# B&R Automation Studio project NAINV104C00R8L515F00 (part 26)

#### Act_Background_Action.st - not listed in the package file held
```iecst
(** 2021-08-01 **)
ACTION Act_Background_Action:
	//Action function
//testing funciton
	IF EDGEPOS(bSimBrdInZone1) THEN
		tyHermesBoardAvailableAttribAddr.udiProductTypeId := p_ProdRcpCurrRcp0Nm;
		tyHermesBoardAvailableAttribAddr.udiWidth  := p_ProdRcpCurrRcp0Width;
		fHermesGenerateBrdAvlDat(ADR(a_tyHermesBrdAvlData[1]),tyHermesBoardAvailableAttribAddr);
		fHermesAddEditAttribBrdAvlDat(ADR(a_tyHermesBrdAvlData[1]),'Action',sSelectedActtoUpdate);
		bSimBrdInZone1 := FALSE;
	END_IF
	IF EDGEPOS(bSimBrdInZone2) THEN
		tyHermesBoardAvailableAttribAddr.udiProductTypeId := p_ProdRcpCurrRcp0Nm;
		tyHermesBoardAvailableAttribAddr.udiWidth  := p_ProdRcpCurrRcp0Width;
		fHermesGenerateBrdAvlDat(ADR(a_tyHermesBrdAvlData[2]),tyHermesBoardAvailableAttribAddr);
		fHermesAddEditAttribBrdAvlDat(ADR(a_tyHermesBrdAvlData[2]),'Action',sSelectedActtoUpdate);
		bSimBrdInZone2 := FALSE;
	END_IF
	IF EDGEPOS(bSimBrdInZone3) THEN
		tyHermesBoardAvailableAttribAddr.udiProductTypeId := p_ProdRcpCurrRcp0Nm;
		tyHermesBoardAvailableAttribAddr.udiWidth  := p_ProdRcpCurrRcp0Width;
		fHermesGenerateBrdAvlDat(ADR(a_tyHermesBrdAvlData[3]),tyHermesBoardAvailableAttribAddr);
		fHermesAddEditAttribBrdAvlDat(ADR(a_tyHermesBrdAvlData[3]),'Action',sSelectedActtoUpdate);
		bSimBrdInZone3 := FALSE;
	END_IF
//	IF EDGEPOS(bSimSearch) THEN
//		testresult1 := fHermesSrchAttribValueBrdAvlDat(ADR(a_tyHermesBrdAvlData[1]),'Action',ADR(sAttribReadValue));
//	END_IF
//	IF EDGEPOS(bSimDelete) THEN
//		testresult2 := fHermesDeleteAttribBrdAvlDat(ADR(a_tyHermesBrdAvlData[1]),'Action');
//	END_IF

	IF EDGEPOS(bSimShiftBoardFoward) THEN
		memmove(ADR(a_tyHermesBrdAvlData[endpos]),ADR(a_tyHermesBrdAvlData[startpos]),SIZEOF(a_tyHermesBrdAvlData[startpos]));
		memset(ADR(a_tyHermesBrdAvlData[startpos]),0,SIZEOF(a_tyHermesBrdAvlData[startpos]));
		memmove(ADR(a_bLinkOpsGConvHvBrd[endpos]),ADR(a_bLinkOpsGConvHvBrd[startpos]),SIZEOF(a_bLinkOpsGConvHvBrd[startpos]));
		memset(ADR(a_bLinkOpsGConvHvBrd[startpos]),0,SIZEOF(a_bLinkOpsGConvHvBrd[startpos]));
	END_IF
	IF EDGEPOS(bSimClear) THEN
		memset(ADR(a_tyHermesBrdAvlData[dltpos]),0,SIZEOF(a_tyHermesBrdAvlData[dltpos]));
	END_IF
//end of testing

//	In state Below
//	Zone[supported action]    0 | 1 | 2
//	Brd(supported action)    A | B | C

	FOR usiZone := usiZoneSupported TO 1 BY -1 DO
		//assiging action
		//update for next machine or zone action
		IF  NOT(a_bUIZonePause[usiZone]) THEN
			a_bBlkDSForAction[usiZone] := FALSE;
			a_bUIPromptActionSelect[usiZone] := FALSE;
		ELSE
			a_bBlkDSForAction[usiZone] := TRUE;
			IF EDGEPOS(a_bOpsDsStandByStep[usiZone]) THEN
				a_bUIPromptActionSelect[usiZone] := TRUE ;
			END_IF

			IF EDGENEG(a_bUIPromptActionSelect[usiZone])  THEN
				a_bUIZonePause[usiZone] := FALSE;
				udiSelectedModtoUpt := a_eModSelectedforCurrZone[usiZone];
				sSelectedActtoUpdate := UDINT_TO_STRING(udiSelectedModtoUpt);
				fHermesAddEditAttribBrdAvlDat(ADR(a_tyHermesBrdAvlData[usiZone]),'Action',sSelectedActtoUpdate);

			END_IF
		END_IF

		//switch the mod for that zone as soon as possible
		//below for preparing action for unoccupied zone starting from right most

		//1)block zone occurred to prevent the middle zone stop reacting to the pending board which does not meet its supported action
		//2)not until the estimated board reach the supported zone, the other left zone will not assigned with action
		//3)compare the leftblock , if reservation zone and occupied zone happened at same time, choose the leftmost zone
		IF usiZone = usiZoneSupported THEN
			usiLeftmostBlockedZone := usiZone;
		ELSIF usiZone < usiLeftmostBlockedZone THEN
			usiLeftmostBlockedZone := usiZone; //check the left block zone
		END_IF

		IF a_bLinkOpsGConvStepInitDone[usiZone] THEN
			IF NOT(a_bLinkOpsGConvHvBrd[usiZone]) THEN
				memset(ADR(a_tyActionReservedForZone[usiZone]),0,SIZEOF(a_tyActionReservedForZone[usiZone]));
				IF usiLeftmostBlockedZone <> 0 THEN //occured there is zone reserved or occupied at zone 1
					FOR usiBrdZone := usiLeftmostBlockedZone TO 1 BY -1 DO
						IF a_bLinkOpsGConvHvBrd[usiBrdZone] THEN
							IF (usiBrdZone-1) < usiZone THEN
								usiLeftmostBlockedZone :=  usiBrdZone; //current board position as limit
							END_IF
							iActionAttributeIdx := fHermesSrchAttribValueBrdAvlDat(ADR(a_tyHermesBrdAvlData[usiBrdZone]),'Action',ADR(sAttribReadValue));
							IF iActionAttributeIdx <> -1 THEN
								iActionOnBrd := STRING_TO_INT(sAttribReadValue);
								IF iActionOnBrd <> 0 AND (1 <= iActionOnBrd  AND iActionOnBrd <= usiMaxActionSupported )THEN
									IF tbActionSupportedByZone[usiZone,iActionOnBrd] THEN
										fHermesSrchAttribValueBrdAvlDat(ADR(a_tyHermesBrdAvlData[usiBrdZone]),'BoardId',ADR(sAttribReadValue));
										//the zone pro-react to action on board
										IF (usiBrdZone-1) < usiZone THEN
											usiLeftmostBlockedZone := usiBrdZone -1; //choose board starting from left side
										END_IF
										a_tyActionReservedForZone[usiZone].iAction := iActionOnBrd; //found support on this zone
										a_tyActionReservedForZone[usiZone].iAttributeIdx := iActionAttributeIdx +1;
										a_tyActionReservedForZone[usiZone].sBoardId := sAttribReadValue;
										EXIT;
									END_IF
								END_IF
							END_IF
							IF a_tyActionReservedForZone[usiZone].iAction <> iActionOnBrd OR iActionOnBrd = 0 THEN
								EXIT; //when non-supported board stuck at middle then do no consider further
							END_IF
						END_IF
					END_FOR
				END_IF
			ELSE // if have board
				IF (usiZone -1) < usiLeftmostBlockedZone THEN
					usiLeftmostBlockedZone := usiZone -1;
				END_IF
				//update when action completed
				fHermesSrchAttribValueBrdAvlDat(ADR(a_tyHermesBrdAvlData[usiZone]),'BoardId',ADR(sAttribReadValue));
				IF a_tyActionReservedForZone[usiZone].iAction <> 0 AND sAttribReadValue =  a_tyActionReservedForZone[usiZone].sBoardId THEN
					IF a_tyActionReservedForZone[usiZone].bActionCompl THEN
						a_tyHermesBrdAvlData[usiZone].a_tyXMLTableDataBrdAvl[a_tyActionReservedForZone[usiZone].iAttributeIdx].sValue	:= '0';
					END_IF
				ELSE //refind an action for the board in current zone
					memset(ADR(a_tyActionReservedForZone[usiZone]),0,SIZEOF(a_tyActionReservedForZone[usiZone]));
					iActionAttributeIdx := fHermesSrchAttribValueBrdAvlDat(ADR(a_tyHermesBrdAvlData[usiZone]),'Action',ADR(sAttribReadValue));
					IF iActionAttributeIdx <> -1 THEN
						iActionOnBrd := STRING_TO_INT(sAttribReadValue);
						IF iActionOnBrd <> 0 AND (1 <= iActionOnBrd  AND iActionOnBrd <= usiMaxActionSupported )THEN
							IF tbActionSupportedByZone[usiZone,iActionOnBrd] THEN
								//react
								fHermesSrchAttribValueBrdAvlDat(ADR(a_tyHermesBrdAvlData[usiZone]),'BoardId',ADR(sAttribReadValue));
								a_tyActionReservedForZone[usiZone].iAction := iActionOnBrd; //found support on this zone
								a_tyActionReservedForZone[usiZone].iAttributeIdx := iActionAttributeIdx +1;
								a_tyActionReservedForZone[usiZone].sBoardId := sAttribReadValue;
								EXIT;
							END_IF
						END_IF
					END_IF
				END_IF
			END_IF

		END_IF

	END_FOR

END_ACTION
```

### USHermes.var - Change By Project
```iecst
(*2020-09-10*)
(**)
(*Action & State & Status*)
VAR
	p_USHermesStat : UDINT;
	p_USHermesStatus : UDINT;
	p_USHermesStatTxt : UDINT;
END_VAR
(**)
(*Alarm*)
VAR
	p_USHermesAlmData : UDINT;
	p_USHermesAlmData1 : UDINT;
	p_USHermesAlmData2 : UDINT;
	p_USHermesAlmData3 : UDINT;
	p_USHermesAlmData4 : UDINT;
	p_USHermesAlmData5 : UDINT;
	p_USHermesInfoData : UDINT;
END_VAR
(**)
(*Output*)
VAR
	p_USHermesTableDataBrdAvl : UDINT;
	p_USHermesTableDataBrdAvlTtlIdx : UDINT;
	p_USHermesConnected : UDINT;
	p_USHermesHandshakeDone : UDINT;
	p_USHermesAccDataReq : UDINT;
	p_USHermesOverWriteSlt : UDINT;
	p_USHermesOverWriteWidth : UDINT;
	p_USHermesReqRecipeNm : UDINT;
	p_USHermesReqWidthInUM : UDINT;
	p_USHermesReqMinSltValue : UDINT;
	p_USHermesReqMaxSltValue : UDINT;
	p_USHermesReqPitch : UDINT;
	p_USHermesUSRdy : UDINT;
	p_USHermesDSRdy : UDINT;
	p_USHermesUSGdRdy : UDINT;
	p_USHermesDSGdRdy : UDINT;
	p_USHermesTransporting : UDINT;
	p_USHermesStopTransport : UDINT;
	p_USHermesBlkUS : UDINT;
	p_USHermesInternalSnd : UDINT;
	p_USHermesAccDataMnl : UDINT;
	p_USHermesStopTransportSnd : UDINT;
	p_USHermestyBoardAvailable : UDINT;
	p_USHermesBoardArrivedData : UDINT;
	p_USHermesRcvBoardInfoOk : UDINT;
	p_USHermesRcvbBoardInfoIncompl : UDINT;
	p_USHermesBoardInfoData : UDINT;
	p_USHermesCommandParam : UDINT;
	p_USHermesReverseDSSendBFId : UDINT;
	p_USHermesProcessRouteTrigger : UDINT;
	p_USHermesAction : UDINT;
	p_USHermesBrdForecastRcv : UDINT;
	p_USHermesBoardAvailableRcved : UDINT;
	p_USHermesStopTransportSent : UDINT;
	p_USHermesStopTransportSentMsg : UDINT;
	p_USHermesBrdForecast : UDINT;
END_VAR
```

### Program Logical/Hermes/USHermes (IEC, version 1.00.0) - 1.00.0 - NtHermes v5.00.0 , NtTCP v5.00.0 , NtMessage v5.00.0

#### Init.st - Change By Project
```iecst
(** 2020-09-10 **)
PROGRAM _INIT

	(* Always Change If Project Change *)

	//Pass Address To Global Address For External Use
	//Action, State & Status
	p_USHermesStat		:= ADR(eStat);
	p_USHermesStatus	:= ADR(eMainStatus);
	p_USHermesStatTxt	:= ADR(sStatTxt);

	//Alarm
	p_USHermesAlmData	:= ADR(tyAlmData);
	p_USHermesAlmData1	:= ADR(tyAlmData1);
	p_USHermesAlmData2	:= ADR(tyAlmData2);
	p_USHermesAlmData3	:= ADR(tyAlmData3);
	p_USHermesAlmData4	:= ADR(tyAlmData4);
	p_USHermesAlmData5	:= ADR(tyAlmData5);
	p_USHermesInfoData	:= ADR(tyInfoData);

	//Output
	p_USHermesTableDataBrdAvl		:= ADR(a_tyXMLTableDataBrdAvl);
	p_USHermesTableDataBrdAvlTtlIdx	:= ADR(iXMLTableDataBrdAvlTtlIdx);
	p_USHermesConnected				:= ADR(bConnected);
	p_USHermesHandshakeDone			:= ADR(bHandshakeDone);
	p_USHermesAccDataReq			:= ADR(bAccDataReq);
	p_USHermesOverWriteSlt			:= ADR(bOverWriteSlt);
	p_USHermesOverWriteWidth		:= ADR(bOverWriteWidth);
	p_USHermesReqRecipeNm			:= ADR(sReqRecipeNm);
	p_USHermesReqWidthInUM			:= ADR(diReqWidthInUM);
	p_USHermesReqMinSltValue		:= ADR(diReqMinSltValue);
	p_USHermesReqMaxSltValue		:= ADR(diReqMaxSltValue);
	p_USHermesReqPitch				:= ADR(diReqPitch);
	p_USHermesUSRdy					:= ADR(bUSRdy);
	p_USHermesDSRdy					:= ADR(bDSRdy);
	p_USHermesUSGdRdy				:= ADR(bUSGdRdy);
	p_USHermesDSGdRdy				:= ADR(bDSGdRdy);
	p_USHermesTransporting			:= ADR(bTransporting);
	p_USHermesStopTransport			:= ADR(bStopTransport);
	p_USHermesBlkUS					:= ADR(bBlkUS);
	p_USHermesInternalSnd			:= ADR(sInternalSnd);
	p_USHermesAccDataMnl			:= ADR(bAccDataMnl);
	p_USHermesStopTransportSnd 		:= ADR(bStopTransportSnd);

	p_USHermestyBoardAvailable		:= ADR(tyBoardAvailableRcv);
	p_USHermesRcvBoardInfoOk        := ADR(bRcvBoardInfoOk);
	p_USHermesRcvbBoardInfoIncompl  := ADR(bRcvBoardInfoIncompl);
	p_USHermesBoardInfoData         := ADR(tySendBoardInfoAcc); //Pass "SendBoardInfo" data for DSHermes "BoardAvailable", for inserted PCB
	p_USHermesBoardArrivedData		:= ADR(tyBoardArrivedInfo); //"BoardArrived" data for SupervisoryHermes

	//command

	p_USHermesCommandParam			:= ADR(tyCommandParam);

	//Calling  on Reverse DS
	p_USHermesReverseDSSendBFId		:= ADR(bReverseDSSndBfWBrdID);
	p_USHermesProcessRouteTrigger	:= ADR(bTriggerUpdateRoute);

	//Action
	p_USHermesAction				:= ADR(iAction);

	//p_USHermesSwitchtoReverseReceive 	:= ADR(bSwitchtoReverseReceive);
	(* Always Change If Project Change *)

	p_USHermesBrdForecast			:= ADR(tyBoardForecastRcv);
	p_USHermesBrdForecastRcv 		:= ADR(bBrdForecastRcv);
	p_USHermesStopTransportSent    	:= ADR(bStopTransportSent);
	p_USHermesStopTransportSentMsg  := ADR(tyStopTransport);
	p_USHermesBoardAvailableRcved   :=ADR(bBoardAvailableRcved);
END_PROGRAM
```

#### Act_InitGlobal.st - Change By Project
```iecst
(** 2019-06-28 **)
ACTION Act_InitGlobal:

	(* Always Change If Project Change *)

	//Pass Data To Link
	p_bLinkStartupRun ACCESS p_StartupRun;
	p_eLinkMcParamUSCommMod ACCESS p_McParamUSCommMod;

	p_eLinkConvDir ACCESS p_NtParamProjConvDir;
	p_bLinkDILeftSen ACCESS p_DIConvLftSen;
	p_bLinkDIRightSen ACCESS p_DIConvRgtSen;

	p_bLinkOpsInvertStepInitDone ACCESS p_OpsInvertStepInitDone;
	p_bLinkOpsRun ACCESS p_OpsRun;

	//Pass Data To Internal Use
	p_udiRstErr ACCESS p_RstErrReset;
	p_bPrep ACCESS p_NtParamHermesPrep;
	p_tyParam ACCESS p_HermesUSParam1;
	p_sIPAddr ACCESS p_HWInfoIPAddr;
	p_tyDTStructure ACCESS p_TimeCurrDTStruct;
	p_dtCurrDT ACCESS p_TimeCurrDT;
	p_sMcId ACCESS p_McParamMcNm;
	p_sRecipeNm ACCESS p_ProdRcpCurrRcp0Nm;
	p_diWidthInUM ACCESS p_ProdRcpCurrRcp0Width;
	p_udiAliveIdleTimeInSec ACCESS p_NtParamUSHermesAliveTmInSec;
	p_tConnTimeOut ACCESS p_NtParamUSHermesConnTO;
	p_diTransferInTO ACCESS p_McParamTranInErrDlyTm;
	p_bInterruptSen ACCESS p_DIConvLftSen;
	p_bOpsRun ACCESS p_OpsRun;
	p_udiFileKeepDay ACCESS p_NtParamUSHermesFileKeepDay;
	p_sProgNm ACCESS p_NtParamUSHermesProgNm;
	p_bNtSettingsLoadDone ACCESS p_StartupNtSettingsLoadDone;
	p_bAccDataRdy ACCESS p_USHermesUSRdy;
	p_sRmtMcId ACCESS p_RmtHermesCurrentConfMcId;
	p_bRmtPrep ACCESS p_NtParamHermesRmtPrep;
	p_bRmtEn ACCESS p_McParamHermesRmtEn;
	pa_tyProdRcpList ACCESS p_ProdRcpCurrList;
	p_tyProdRcpCurrRcp ACCESS p_ProdRcpCurrRcp0;
	p_bMcParamMnlAccData ACCESS p_McParamMnlAccDat;
	p_bUIAccData ACCESS p_UIProdAccData;

	pa_tyHermesDSParam ACCESS pa_HermesDSParam;

	p_bHermesSwitchtoRvrseTransport ACCESS p_HermesSwitchtoReverseTransport;//p_USHermes2SwitchtoReverseRcv;
	//Query Board Info
	p_bTransportFinished ACCESS p_DSHermesTransportFinish ;
	p_bQueryBoardInfo ACCESS p_UIQueryBoardInfo;
	p_bManualInsertZoneHvBrd ACCESS p_ConvHvBrd; //insert zone (can input conv or ouput conv)
	p_bManualInsertEndSen ACCESS p_DIConvRgtSen;
	p_bConvHvBrd ACCESS p_ConvHvBrd; //first zone
	//Reverse Machine Ready
	//p_bReceiveReverseUSMcRdy ACCESS p_DSHermes2RcvReverseUSMcRdy;

	(* Always Change If Project Change *)

END_ACTION
```

#### InputRef_Link.var - Change By Project
```iecst
(*2019-06-04*)
(**)
VAR
	p_bLinkStartupRun : REFERENCE TO BOOL;
	p_eLinkMcParamUSCommMod : REFERENCE TO eMcSetCommMod;
	bHermesRun : BOOL;
	bHermesStop : BOOL;
END_VAR
(**)
VAR
	p_eLinkConvDir : REFERENCE TO eConvDir;
	p_bLinkDILeftSen : REFERENCE TO BOOL;
	p_bLinkDIRightSen : REFERENCE TO BOOL;
	pa_tyLinkProdRcpList : REFERENCE TO ARRAY[1..c_udiProdRcpMax] OF tyProdRcpParam;
	p_tyLinkProdRcpCurrRcp : REFERENCE TO tyProdRcpParam;
	p_bLinkMcParamMnlAccData : REFERENCE TO BOOL;
	p_bLinkOpsStop : REFERENCE TO BOOL;
	p_bLinkUIAccData : REFERENCE TO BOOL;
	sWidthInUMTemp : STRING[80];
END_VAR
(**)
VAR
	p_bLinkConvHvBrd : REFERENCE TO BOOL;
	p_bLinkOpsRun : REFERENCE TO BOOL;
	p_bLinkOpsInvertStepInitDone : REFERENCE TO BOOL;
END_VAR
(**)
VAR
	fbDlyTmr : TON := (PT:=T#5s);
	fbDeleteLogTmr : TON := (PT:=T#24h);
END_VAR
```

#### Act_LinkEn.st - Change By Project
```iecst
(** 2019-03-15 **)
ACTION Act_LinkEn:

	//Link bPrep, bEn & bDis

END_ACTION
```

#### Act_Link.st - Change By Project
```iecst
(** 2019-06-04 **)
ACTION Act_Link:

	//Receive Alive Time
	p_tyParam.tRcvAlive	:= p_tyParam.tSndAlive * 2;

	//Transfer Complete
	IF (p_eLinkConvDir = ConvDirLToR) OR (p_eLinkConvDir = ConvDirLToL) THEN
		p_bRcvCompl	:= EDGENEG(p_bLinkDILeftSen);
	ELSE
		p_bRcvCompl	:= EDGENEG(p_bLinkDIRightSen);
	END_IF

	//Ready Receive
	p_bRdyRcv ACCESS p_OpsInvertStepUSCommTmr;

	//Ready Transport
	p_bRdyTransport	:= TRUE;

	//Accept New Recipe Condition
	p_bAccNewRcpCond	:= p_bLinkOpsRun = TRUE;

	//Routing
	p_bProcessRouteEn := p_bManualRmvRoute OR p_bReturnRoute OR p_bNomRouteEn;

END_ACTION
```

#### Cyclic.st - Do Not Change!!!
```iecst
(** 2020-09-10 **)
PROGRAM _CYCLIC

	IF bInitDone = FALSE THEN
		bInitDone	:= TRUE;

		Act_InitLocal;
		Act_InitGlobal;

	ELSIF bInitialDone = FALSE THEN
		IF p_bNtSettingsLoadDone = TRUE THEN
			bInitialDone	:= TRUE;

			Act_Initial;
		END_IF

	ELSE

		Act_RstErr;
		Act_LinkAction;
		Act_Action;
		Act_LinkEn;

		IF (p_bPrep = TRUE) AND (p_bEn = TRUE) AND (p_bDis = FALSE) THEN

			Act_Link;
			Act_Main;
			Act_Background;
		ELSE
			Act_Main_Disable;

			IF eStat <> HermesActIdle THEN
				eStatus	:= Done;
			ELSE
				eStatus	:= Idle;
			END_IF
		END_IF

		Act_CombineErr;
		Act_Alarm;
		Act_Alarm1;
		Act_Alarm2;
		Act_Alarm3;
		Act_Alarm4;
		Act_Alarm5;

	END_IF

END_PROGRAM
```

#### Act_RstErr.st - Do Not Change!!!
```iecst
(** 2019-03-15 **)
ACTION Act_RstErr:

	IF p_udiRstErr <> udiRstErrOld THEN
		bRstErr			:= TRUE;
		udiRstErrOld	:= p_udiRstErr;
	ELSE
		bRstErr			:= FALSE;
	END_IF

END_ACTION
```

#### Act_InitLocal.st - Do Not Change!!!
```iecst
(** 2019-06-28 **)
ACTION Act_InitLocal:

	//Input Reference Link To Local Variable
	p_eAct ACCESS ADR(eAct);
	p_udiRstErr ACCESS ADR(udiRstErr);
	p_bPrep ACCESS ADR(bPrep);
	p_bEn ACCESS ADR(bEn);
	p_bDis ACCESS ADR(bDis);
	p_tyParam ACCESS ADR(tyParam);
	p_sIPAddr ACCESS ADR(sIPAddr);
	p_tyDTStructure ACCESS ADR(tyDTStructure);
	p_dtCurrDT ACCESS ADR(dtCurrDT);
	p_bRdyRcv ACCESS ADR(bRdyRcv);
	p_bRdyTransport ACCESS ADR(bRdyTransport);
	p_bRcvCompl ACCESS ADR(bRcvCompl);
	p_bRcvIncompl ACCESS ADR(bRcvInCompl);
	p_bRcvNotStart ACCESS ADR(bRcvNotStart);
	p_bBAWidthEn ACCESS ADR(bBAWidthEn);
	p_bBASltEn ACCESS ADR(bBASltEn);
	p_bBFWidthEn ACCESS ADR(bBFWidthEn);
	p_bBFSltEn ACCESS ADR(bBFSltEn);
	p_sMcId ACCESS ADR(sMcId);
	p_sInterfaceId ACCESS ADR(sInterfaceId);
	p_sVersion ACCESS ADR(sVersion);
	p_eFailedBoard ACCESS ADR(eFailedBoard);
	p_sRecipeNm ACCESS ADR(sRecipeNm);
	p_diWidthInUM ACCESS ADR(diWidthInUM);
	p_diMinSltValue ACCESS ADR(diMinSltValue);
	p_diMaxSltValue ACCESS ADR(diMaxSltValue);
	p_diPitch ACCESS ADR(diPitch);
	p_diTtlSlt ACCESS ADR(diTtlSlt);
	p_diSltToSltInUM ACCESS ADR(diSltToSltInUM);
	p_udiSndBffrSize ACCESS ADR(udiSndBffrSize);
	p_udiRcvBffrSize ACCESS ADR(udiRcvBffrSize);
	p_udiAliveIdleTimeInSec ACCESS ADR(udiAliveIdleTimeInSec);
	p_tConnTimeOut ACCESS ADR(tConnTimeOut);
	p_diTransferInTO ACCESS ADR(diTransferInTO);
	p_bOpsRun ACCESS ADR(bOpsRun);
	p_bInterruptSen ACCESS ADR(bInterruptSen);
	p_udiFileKeepDay ACCESS ADR(udiFileKeepDay);
	p_sProgNm ACCESS ADR(sProgNm);
	p_bNtSettingsLoadDone ACCESS ADR(bNtSettingsLoadDone);
	p_bAccDataRdy ACCESS ADR(bAccDataRdy);
	p_sRmtMcId ACCESS ADR(sRmtMcId);
	p_bRmtPrep ACCESS ADR(bRmtPrep);
	p_bRmtEn ACCESS ADR(bRmtEn);
	p_bAccNewRcpCond ACCESS ADR(bAccNewRcpCond);
	p_sInfoMsg ACCESS ADR(sInfoMsg);
	p_sInfoMsg1 ACCESS ADR(sInfoMsg1);
	p_sInfoMsg2 ACCESS ADR(sInfoMsg2);
	p_bInternalUse ACCESS ADR(bInternalUse);
	p_sInternalRcv ACCESS ADR(sInternalRcv);
	pa_tyProdRcpList ACCESS ADR(a_tyProdRcpList);
	p_tyProdRcpCurrRcp ACCESS ADR(tyProdRcpCurrRcp);
	p_bMcParamMnlAccData ACCESS ADR(bMcParamMnlAccData);
	p_bUIAccData ACCESS ADR(bUIAccData);

	p_tyDSHermesCurrBASnd ACCESS ADR(tyBoardAvailableDummy);

	p_bManualRmvRoute ACCESS ADR(bManualRmvRoute);
	p_bReturnRoute ACCESS ADR(bReturnRoute);
	p_bNomRouteEn ACCESS ADR(bNomRouteEn);
	p_bProcessRouteEn ACCESS ADR(bProcessRouteEn);

	p_bReverseReceiveRoute ACCESS ADR(bReverseReceiveRoute);
	p_bReceiveReverseUSMcRdy ACCESS ADR(bReceiveReverseUSMcRdy);

	p_sTopBarcode  ACCESS ADR(sUITopBarcode);
	p_sBottomBarcode ACCESS ADR(sUIBottomBarcode);
END_ACTION
```

#### Act_Action.st - Do Not Change!!!
```iecst
(** 2019-03-25 **)
ACTION Act_Action:

	//Reset Error
	IF (eStatus = Error) AND bRstErr THEN
		p_eAct	:= HermesActIdle;
		eStat	:= HermesActIdle;
	END_IF

	//Set p_eAct
	IF eStatus = Idle OR eStatus = Done THEN // OR eStatus = Busy
		eStat	:= p_eAct;
	END_IF

END_ACTION
```

#### Act_Main.st - Do Not Change!!!
```iecst
(** 2019-04-08 **)
ACTION Act_Main:

	IF eStatOld <> eStat THEN
		fbFileOldDel1(bEn := FALSE);

		sStatTxt	:= a_sStatText[eStat];

		eStatOld	:= eStat;

		eStatus		:= Busy;
	END_IF

	//Main
	CASE eStat OF

		HermesActIdle:
			eStatus	:= Idle;

		HermesActBGStartRun:
			IF eStatus = Idle OR eStatus = Busy THEN

				bRun	:= TRUE;
				bStop	:= FALSE;
				eStatus	:= Done;

			END_IF

		HermesActBGStopRun:
			IF eStatus = Idle OR eStatus = Busy THEN

				bStop	:= TRUE;
				eStatus	:= Done;

			END_IF

		HermesActDeleteOldLog:
			IF eStatus = Idle OR eStatus = Busy THEN

				eStatus	:= Busy;

				fbFileOldDel1.dtDTNow	:= p_dtCurrDT;
				fbFileOldDel1(bEn := TRUE);
				IF fbFileOldDel1.udiStatus = 0 THEN
					eStatus	:= Done;
				ELSIF fbFileOldDel1.udiStatus < 65534 THEN
					eStatus		:= Error;

					IF fbFileOldDel1.udiStatus = 1910 THEN
						udiStatus	:= 10154;	//Get Directory Info Error While Deleting Old Log
					ELSIF fbFileOldDel1.udiStatus = 1911 THEN
						udiStatus	:= 10155;	//Directory Read Error While Deleting Old Log
					ELSIF fbFileOldDel1.udiStatus = 1912 THEN
						udiStatus	:= 10156;	//File Delete Error While Deleting Old Log
					ELSE
						udiStatus	:= fbFileOldDel1.udiStatus;
					END_IF
				END_IF

			END_IF

		ELSE
			IF eStatus = Idle OR eStatus = Busy THEN
				eStatus	:= Done;
			END_IF

	END_CASE

END_ACTION
```

#### Act_Background_TCPConnect.st - Do Not Change!!!
```iecst
(** 2020-09-10 **)
ACTION Act_Background_TCPConnect:

	IF eStatus1 <> Error AND eStatus2 <> Error THEN

		//Connect Server
		fbClntConnect.sClntIP		:= p_sIPAddr;
		fbClntConnect.sSvrIP		:= p_tyParam.sHostAddress;
		fbClntConnect.uiClntPort	:= p_tyParam.uiClntPort;
		fbClntConnect.uiSvrPort		:= p_tyParam.uiHostPort;
		fbClntConnect(bEn := TRUE);

		IF fbClntConnect.udiStatus = 0 THEN
			udiTCPIdent	:= fbClntConnect.udiTCPIdent;
			fbClntConnect(bEn := FALSE);

		ELSIF fbClntConnect.udiStatus = 2313 THEN
			fbClntConnect(bEn := FALSE);

		ELSIF fbClntConnect.udiStatus = 2323 OR bConnected= FALSE THEN
			udiStatus5	:= 10013;	//Client Connect Time Out Warning

		ELSIF fbClntConnect.udiStatus < 65534 THEN
			eStatus1	:= Error;

			IF fbClntConnect.udiStatus = 2300 THEN
				udiStatus1	:= 10000;	//Invalid Ident While Client Connecting
			ELSIF fbClntConnect.udiStatus = 2302 THEN
				udiStatus1	:= 10001;	//Setting Keep Alive Interval Time Error While Client Connecting
			ELSIF fbClntConnect.udiStatus = 2303 THEN
				udiStatus1	:= 10002;	//Setting Keep Alive Idle Time Error While Client Connecting
			ELSIF fbClntConnect.udiStatus = 2304 THEN
				udiStatus1	:= 10003;	//Setting Keep Alive Count Error While Client Connecting
			ELSIF fbClntConnect.udiStatus = 2305 THEN
				udiStatus1	:= 10004;	//Setting Keep Alive Error While Client Connecting
			ELSIF fbClntConnect.udiStatus = 2306 THEN
				udiStatus1	:= 10005;	//Setting Receive Buffer Error While Client Connecting
			ELSIF fbClntConnect.udiStatus = 2307 THEN
				udiStatus1	:= 10006;	//Setting Send Buffer Error While Client Connecting
			ELSIF fbClntConnect.udiStatus = 2308 THEN
				udiStatus1	:= 10007;	//Setting No Waiting Error While Client Connecting
			ELSIF fbClntConnect.udiStatus = 2309 THEN
				udiStatus1	:= 10008;	//TCP Open Port Error While Client Connecting
			ELSIF fbClntConnect.udiStatus = 2310 THEN
				udiStatus1	:= 10009;	//Closing TCP Error While Client Connecting
			ELSIF fbClntConnect.udiStatus = 2313 THEN
				udiStatus1	:= 10010;	//Server Connection Failed While Client Connecting
			ELSIF fbClntConnect.udiStatus = 2314 THEN
				udiStatus1	:= 10011;	//Ident In Used While Client Connecting
			ELSIF fbClntConnect.udiStatus = 2315 THEN
				udiStatus1	:= 10012;	//Connect To Server Error While Client Connecting

			ELSE
				udiStatus1	:= fbClntConnect.udiStatus;
			END_IF

		END_IF

	END_IF

END_ACTION
```

#### Act_Background_TCPRcv.st - Do Not Change!!!
```iecst
(** 2019-06-10 **)
ACTION Act_Background_TCPRcv:

	IF eStatus1 <> Error THEN

		//Receive Data
		IF p_bInternalUse = FALSE THEN
			fbRcv.udiTCPIdent	:= udiTCPIdent;
			fbRcv(bEn := TRUE);
		ELSE
			sRcv	:= p_sInternalRcv;
		END_IF

		IF (fbRcv.udiStatus = 0) OR ((p_bInternalUse = TRUE) AND (LEN(sRcv) > 0)) THEN

			fLogDTConvert(ADR(sDT) , p_dtCurrDT);
			memset(ADR(a_sLogList[udiLogCntr]) , 0 , SIZEOF(a_sLogList[udiLogCntr]));
			memcpy(ADR(a_sLogList[udiLogCntr]) + LEN(a_sLogList[udiLogCntr]) , ADR(sDT) , LEN(sDT));
			memcpy(ADR(a_sLogList[udiLogCntr]) + LEN(a_sLogList[udiLogCntr]) , ADR('$r$n') , LEN('$r$n'));
			memcpy(ADR(a_sLogList[udiLogCntr]) + LEN(a_sLogList[udiLogCntr]) , ADR('RCV_FRM_US$r$n') , LEN('RCV_FRM_US$r$n'));
			memcpy(ADR(a_sLogList[udiLogCntr]) + LEN(a_sLogList[udiLogCntr]) , ADR(sRcv) , LEN(sRcv));
			memcpy(ADR(a_sLogList[udiLogCntr]) + LEN(a_sLogList[udiLogCntr]) , ADR('$r$n$r$n') , LEN('$r$n$r$n'));

			udiLogCntr	:= udiLogCntr + 1;
			IF udiLogCntr = 11 THEN
				udiLogCntr	:= 1;
			END_IF

			fXMLConvertToTable(ADR(sRcv) , LEN(sRcv) , ADR(a_tyXMLTableDataRcv) , ADR(a_tyXMLTableDataRcv[0].sTitle) , SIZEOF(a_tyXMLTableDataRcv[0].sTitle) , ADR(a_tyXMLTableDataRcv[0].sValue) , SIZEOF(a_tyXMLTableDataRcv[0].sValue) , ADR(a_tyXMLTableDataRcv[0].uiSize) , SIZEOF(a_tyXMLTableDataRcv[0]) , SIZEOF(a_tyXMLTableDataRcv) / SIZEOF(a_tyXMLTableDataRcv[0]) , ADR(udiXMLTableWriteIdx));

			fbParseXMLTable.iTotalIdxWrite	:= UDINT_TO_INT(udiXMLTableWriteIdx);
			fbParseXMLTable;

			IF fbParseXMLTable.tyMsgType.bCheckAlive = TRUE THEN
				tyMsgTypeRcv.bCheckAlive	:= TRUE;
				tyCheckAliveRcv				:= fbParseXMLTable.tyCheckAlive;
			END_IF

			IF fbParseXMLTable.tyMsgType.bCheckAlivePing = TRUE THEN
				tyMsgTypeRcv.bCheckAlivePing	:= TRUE;
				tyCheckAlivePingRcv				:= fbParseXMLTable.tyCheckAlivePing;
			END_IF

			IF fbParseXMLTable.tyMsgType.bCheckAlivePong = TRUE THEN
				tyMsgTypeRcv.bCheckAlivePong	:= TRUE;
				tyCheckAlivePongRcv				:= fbParseXMLTable.tyCheckAlivePong;
			END_IF

			IF fbParseXMLTable.tyMsgType.bServiceDescription = TRUE THEN
				tyMsgTypeRcv.bServiceDescription	:= TRUE;
				tyServiceDescriptionRcv				:= fbParseXMLTable.tyServiceDescription;
			END_IF

			IF fbParseXMLTable.tyMsgType.bNotification = TRUE THEN
				tyMsgTypeRcv.bNotification	:= TRUE;
				tyNotificationRcv			:= fbParseXMLTable.tyNotification;
			END_IF

			IF fbParseXMLTable.tyMsgType.bBoardAvailable = TRUE THEN
				tyMsgTypeRcv.bBoardAvailable	:= TRUE;
				tyBoardAvailableRcv				:= fbParseXMLTable.tyBoardAvailable;

				memset(ADR(a_tyXMLTableDataBrdAvl) , 0 , SIZEOF(a_tyXMLTableDataBrdAvl));
				memcpy(ADR(a_tyXMLTableDataBrdAvl) , ADR(a_tyXMLTableDataRcv) + (fbParseXMLTable.iBoardAvailableFirstIdx * SIZEOF(a_tyXMLTableDataRcv[0])) , (fbParseXMLTable.iBoardAvailableLastIdx - fbParseXMLTable.iBoardAvailableFirstIdx + 1) * SIZEOF(a_tyXMLTableDataRcv[0]));

				iXMLTableDataBrdAvlTtlIdx	:= fbParseXMLTable.iBoardAvailableLastIdx - fbParseXMLTable.iBoardAvailableFirstIdx + 1;

			END_IF

			IF fbParseXMLTable.tyMsgType.bRevokeBoardAvailable = TRUE THEN
				tyMsgTypeRcv.bRevokeBoardAvailable	:= TRUE;
			END_IF

			IF fbParseXMLTable.tyMsgType.bMachineReady = TRUE THEN
				tyMsgTypeRcv.bMachineReady	:= TRUE;
				tyMachineReady				:= fbParseXMLTable.tyMachineReady;
			END_IF

			IF fbParseXMLTable.tyMsgType.bRevokeMachineReady = TRUE THEN
				tyMsgTypeRcv.bRevokeMachineReady	:= TRUE;
			END_IF

			IF fbParseXMLTable.tyMsgType.bStartTransport = TRUE THEN
				tyMsgTypeRcv.bStartTransport	:= TRUE;
				tyStartTransport				:= fbParseXMLTable.tyStartTransport;
			END_IF

			IF fbParseXMLTable.tyMsgType.bStopTransport = TRUE THEN
				tyMsgTypeRcv.bStopTransport	:= TRUE;
				tyStopTransport				:= fbParseXMLTable.tyStopTransport;
			END_IF

			IF fbParseXMLTable.tyMsgType.bTransportFinished = TRUE THEN
				tyMsgTypeRcv.bTransportFinished	:= TRUE;
				tyTransportFinished				:= fbParseXMLTable.tyTransportFinished;
			END_IF

			IF fbParseXMLTable.tyMsgType.bSetConfiguration = TRUE THEN
				tyMsgTypeRcv.bSetConfiguration	:= TRUE;
				tySetConfiguration				:= fbParseXMLTable.tySetConfiguration;
			END_IF

			IF fbParseXMLTable.tyMsgType.bGetConfiguration = TRUE THEN
				tyMsgTypeRcv.bGetConfiguration	:= TRUE;
			END_IF

			IF fbParseXMLTable.tyMsgType.bCurrentConfiguration = TRUE THEN
				tyMsgTypeRcv.bCurrentConfiguration	:= TRUE;
				tyCurrentConfiguration				:= fbParseXMLTable.tyCurrentConfiguration;
			END_IF

			IF fbParseXMLTable.tyMsgType.bBoardForecast = TRUE THEN
				tyMsgTypeRcv.bBoardForecast	:= TRUE;
				tyBoardForecastRcv				:= fbParseXMLTable.tyBoardForecast;
			END_IF

			IF fbParseXMLTable.tyMsgType.bQueryBoardInfo = TRUE THEN
				tyMsgTypeRcv.bQueryBoardInfo	:= TRUE;
				tyQueryBoardInfo				:= fbParseXMLTable.tyQueryBoardInfo;
			END_IF

			IF fbParseXMLTable.tyMsgType.bSendBoardInfo = TRUE THEN
				tyMsgTypeRcv.bSendBoardInfo	:= TRUE;
				tySendBoardInfoRcv				:= fbParseXMLTable.tySendBoardInfo;
			END_IF

			IF fbParseXMLTable.tyMsgType.bCommand = TRUE THEN
				tyMsgTypeRcv.bCommand	:= TRUE;
				tyCommandRcv			:= fbParseXMLTable.tyCommand;
			END_IF

			fbRcv(bEn := FALSE);

			memset(ADR(sRcv) , 0 , SIZEOF(sRcv));

		ELSIF (fbRcv.udiStatus = 2317) AND (p_bInternalUse = FALSE) THEN
			fbRcv(bEn := FALSE);

			memset(ADR(sRcv) , 0 , SIZEOF(sRcv));

		ELSIF (fbRcv.udiStatus = 2316) AND (p_bInternalUse = FALSE) THEN
			bRstConnection	:= TRUE;

			memset(ADR(sRcv) , 0 , SIZEOF(sRcv));

		ELSIF (fbRcv.udiStatus = 2318) AND (p_bInternalUse = FALSE) THEN
			bRstConnection	:= TRUE;

			memset(ADR(sRcv) , 0 , SIZEOF(sRcv));

		ELSIF (fbRcv.udiStatus < 65534) AND (p_bInternalUse = FALSE) THEN
			eStatus1	:= Error;

			IF fbRcv.udiStatus = 2300 THEN
				udiStatus1	:= 10014;	//Invalid Ident While Receiving Data
			ELSIF fbRcv.udiStatus = 2319 THEN
				udiStatus1	:= 10015;	//TCP Receive Data Error While Receiving Data
			ELSE
				udiStatus1	:= fbRcv.udiStatus;
			END_IF

			memset(ADR(sRcv) , 0 , SIZEOF(sRcv));

		END_IF

	END_IF

END_ACTION
```

#### Act_Background_NotificationRcv.st - Do Not Change!!!
```iecst
(** 2019-03-15 **)
ACTION Act_Background_NotificationRcv:

	IF eStatus1 <> Error THEN

		IF tyMsgTypeRcv.bNotification = TRUE THEN
			tyMsgTypeRcv.bNotification	:= FALSE;

			bRstConnection	:= fHermesNotificationRstConn(tyNotificationRcv) OR bRstConnection;
//			bRstState		:= fHermesNotificationRstState(tyNotificationRcv) OR bRstState;

		END_IF

	END_IF

END_ACTION
```

#### Act_Background_IllegalMsg.st - Do Not Change!!!
```iecst
(** 2019-05-04 **)
ACTION Act_Background_IllegalMsg:

	IF eStatus2 <> Error THEN

		udiStatus2	:= fHermesIllegalMsgUS(fbSequenceUS.eState , tyMsgTypeRcv , fbSequenceUS.bBoardAvailable);

		IF udiStatus2 <> 0 THEN
			eStatus2	:= Error;

			IF udiStatus2 = 2770 THEN
				udiStatus2	:= 10016;	//Receive ServiceDescription While Upstream In Not Connected State
			ELSIF udiStatus2 = 2771 THEN
				udiStatus2	:= 10017;	//Receive BoardAvailable While Upstream In Not Connected State
			ELSIF udiStatus2 = 2772 THEN
				udiStatus2	:= 10018;	//Receive RevokeBoardAvailable While Upstream In Not Connected State
			ELSIF udiStatus2 = 2773 THEN
				udiStatus2	:= 10019;	//Receive MachineReady While Upstream In Not Connected State
			ELSIF udiStatus2 = 2774 THEN
				udiStatus2	:= 10020;	//Receive RevokeMachineReady While Upstream In Not Connected State
			ELSIF udiStatus2 = 2775 THEN
				udiStatus2	:= 10021;	//Receive StartTransport While Upstream In Not Connected State
			ELSIF udiStatus2 = 2776 THEN
				udiStatus2	:= 10022;	//Receive StopTransport While Upstream In Not Connected State
			ELSIF udiStatus2 = 2777 THEN
				udiStatus2	:= 10023;	//Receive TransportFinished While Upstream In Not Connected State
			ELSIF udiStatus2 = 2778 THEN
				udiStatus2	:= 10024;	//Receive BoardForecast While Upstream In Not Connected State
			ELSIF udiStatus2 = 2779 THEN
				udiStatus2	:= 10025;	//Receive BoardAvailable While Upstream In Service Description State
			ELSIF udiStatus2 = 2780 THEN
				udiStatus2	:= 10026;	//Receive RevokeBoardAvailable While Upstream In Service Description State
			ELSIF udiStatus2 = 2781 THEN
				udiStatus2	:= 10027;	//Receive MachineReady While Upstream In Service Description State
			ELSIF udiStatus2 = 2782 THEN
				udiStatus2	:= 10028;	//Receive RevokeMachineReady While Upstream In Service Description State
			ELSIF udiStatus2 = 2783 THEN
				udiStatus2	:= 10029;	//Receive StartTransport While Upstream In Service Description State
			ELSIF udiStatus2 = 2784 THEN
				udiStatus2	:= 10030;	//Receive StopTransport While Upstream In Service Description State
			ELSIF udiStatus2 = 2785 THEN
				udiStatus2	:= 10031;	//Receive TransportFinished While Upstream In Service Description State
			ELSIF udiStatus2 = 2786 THEN
				udiStatus2	:= 10032;	//Receive BoardForecast While Upstream In Service Description State
			ELSIF udiStatus2 = 2787 THEN
				udiStatus2	:= 10033;	//Receive ServiceDescription While Upstream In Not Available Not Ready State
			ELSIF udiStatus2 = 2788 THEN
				udiStatus2	:= 10034;	//Receive RevokeBoardAvailable While Upstream In Not Available Not Ready State
			ELSIF udiStatus2 = 2789 THEN
				udiStatus2	:= 10035;	//Receive MachineReady While Upstream In Not Available Not Ready State
			ELSIF udiStatus2 = 2790 THEN
				udiStatus2	:= 10036;	//Receive RevokeMachineReady While Upstream In Not Available Not Ready State
			ELSIF udiStatus2 = 2791 THEN
				udiStatus2	:= 10037;	//Receive StartTransport While Upstream In Not Available Not Ready State
			ELSIF udiStatus2 = 2792 THEN
				udiStatus2	:= 10038;	//Receive StopTransport While Upstream In Not Available Not Ready State
			ELSIF udiStatus2 = 2793 THEN
				udiStatus2	:= 10039;	//Receive TransportFinished While Upstream In Not Available Not Ready State
			ELSIF udiStatus2 = 2794 THEN
				udiStatus2	:= 10040;	//Receive ServiceDescription While Upstream In Board Available State
			ELSIF udiStatus2 = 2795 THEN
				udiStatus2	:= 10041;	//Receive BoardAvailable While Upstream In Board Available State
			ELSIF udiStatus2 = 2796 THEN
				udiStatus2	:= 10042;	//Receive MachineReady While Upstream In Board Available State
			ELSIF udiStatus2 = 2797 THEN
				udiStatus2	:= 10043;	//Receive RevokeMachineReady While Upstream In Board Available State
			ELSIF udiStatus2 = 2798 THEN
				udiStatus2	:= 10044;	//Receive StartTransport While Upstream In Board Available State
			ELSIF udiStatus2 = 2799 THEN
				udiStatus2	:= 10045;	//Receive StopTransport While Upstream In Board Available State
			ELSIF udiStatus2 = 2800 THEN
				udiStatus2	:= 10046;	//Receive TransportFinished While Upstream In Board Available State
			ELSIF udiStatus2 = 2801 THEN
				udiStatus2	:= 10047;	//Receive BoardForecast While Upstream In Board Available State
			ELSIF udiStatus2 = 2802 THEN
				udiStatus2	:= 10048;	//Receive ServiceDescription While Upstream In Machine Ready State
			ELSIF udiStatus2 = 2803 THEN
				udiStatus2	:= 10049;	//Receive RevokeBoardAvailable While Upstream In Machine Ready State
			ELSIF udiStatus2 = 2804 THEN
				udiStatus2	:= 10050;	//Receive MachineReady While Upstream In Machine Ready State
			ELSIF udiStatus2 = 2805 THEN
				udiStatus2	:= 10051;	//Receive RevokeMachineReady While Upstream In Machine Ready State
			ELSIF udiStatus2 = 2806 THEN
				udiStatus2	:= 10052;	//Receive StartTransport While Upstream In Machine Ready State
			ELSIF udiStatus2 = 2807 THEN
				udiStatus2	:= 10053;	//Receive StopTransport While Upstream In Machine Ready State
			ELSIF udiStatus2 = 2808 THEN
				udiStatus2	:= 10054;	//Receive TransportFinished While Upstream In Machine Ready State
			ELSIF udiStatus2 = 2809 THEN
				udiStatus2	:= 10055;	//Receive ServiceDescription While Upstream In Available And Ready State
			ELSIF udiStatus2 = 2810 THEN
				udiStatus2	:= 10056;	//Receive BoardAvailable While Upstream In Available And Ready State
			ELSIF udiStatus2 = 2811 THEN
				udiStatus2	:= 10057;	//Receive MachineReady While Upstream In Available And Ready State
			ELSIF udiStatus2 = 2812 THEN
				udiStatus2	:= 10058;	//Receive RevokeMachineReady While Upstream In Available And Ready State
			ELSIF udiStatus2 = 2813 THEN
				udiStatus2	:= 10059;	//Receive StartTransport While Upstream In Available And Ready State
			ELSIF udiStatus2 = 2814 THEN
				udiStatus2	:= 10060;	//Receive StopTransport While Upstream In Available And Ready State
			ELSIF udiStatus2 = 2815 THEN
				udiStatus2	:= 10061;	//Receive TransportFinished While Upstream In Available And Ready State
			ELSIF udiStatus2 = 2816 THEN
				udiStatus2	:= 10062;	//Receive BoardForecast While Upstream In Available And Ready State
			ELSIF udiStatus2 = 2817 THEN
				udiStatus2	:= 10063;	//Receive ServiceDescription While Upstream In Transporting State
			ELSIF udiStatus2 = 2818 THEN
				udiStatus2	:= 10064;	//Receive Twice Board Available While Upstream In Transporting State
			ELSIF udiStatus2 = 2819 THEN
				udiStatus2	:= 10065;	//Receive RevokeBoardAvailable Without BoardAvailable While Upstream In Transporting State
			ELSIF udiStatus2 = 2820 THEN
				udiStatus2	:= 10066;	//Receive MachineReady While Upstream In Transporting State
			ELSIF udiStatus2 = 2821 THEN
				udiStatus2	:= 10067;	//Receive RevokeMachineReady While Upstream In Transporting State
			ELSIF udiStatus2 = 2822 THEN
				udiStatus2	:= 10068;	//Receive StartTransport While Upstream In Transporting State
			ELSIF udiStatus2 = 2823 THEN
				udiStatus2	:= 10069;	//Receive StopTransport While Upstream In Transporting State
			ELSIF udiStatus2 = 2824 THEN
				udiStatus2	:= 10070;	//Receive ServiceDescription While Upstream In Transport Finished State
			ELSIF udiStatus2 = 2825 THEN
				udiStatus2	:= 10071;	//Receive BoardAvailable While Upstream In Transport Finished State
			ELSIF udiStatus2 = 2826 THEN
				udiStatus2	:= 10072;	//Receive RevokeBoardAvailable While UpstreamWhile Upstream In Transport Finished State
			ELSIF udiStatus2 = 2827 THEN
				udiStatus2	:= 10073;	//Receive MachineReady While Upstream In Transport Finished State
			ELSIF udiStatus2 = 2828 THEN
				udiStatus2	:= 10074;	//Receive RevokeMachineReady While Upstream In Transport Finished State
			ELSIF udiStatus2 = 2829 THEN
				udiStatus2	:= 10075;	//Receive StartTransport While Upstream In Transport Finished State
			ELSIF udiStatus2 = 2830 THEN
				udiStatus2	:= 10076;	//Receive TransportFinished While Upstream In Transport Finished State
			ELSIF udiStatus2 = 2831 THEN
				udiStatus2	:= 10077;	//Receive StopTransport While Upstream In Transport Finished State
			ELSIF udiStatus2 = 2832 THEN
				udiStatus2	:= 10078;	//Receive BoardForecast While Upstream In Transport Finished State
			ELSIF udiStatus2 = 2833 THEN
				udiStatus2	:= 10079;	//Receive ServiceDescription While Upstream In Transport Stopped State
			ELSIF udiStatus2 = 2834 THEN
				udiStatus2	:= 10080;	//Receive Twice Board Available While Upstream In Transport Stopped State
			ELSIF udiStatus2 = 2835 THEN
				udiStatus2	:= 10081;	//Receive RevokeBoardAvailable Without BoardAvailable While Upstream In Transport Stopped State
			ELSIF udiStatus2 = 2836 THEN
				udiStatus2	:= 10082;	//Receive MachineReady While Upstream In Transport Stopped State
			ELSIF udiStatus2 = 2837 THEN
				udiStatus2	:= 10083;	//Receive RevokeMachineReady While Upstream In Transport Stopped State
			ELSIF udiStatus2 = 2838 THEN
				udiStatus2	:= 10084;	//Receive StartTransport While Upstream In Transport Stopped State
			ELSIF udiStatus2 = 2839 THEN
				udiStatus2	:= 10085;	//Receive StopTransport While Upstream In Transport Stopped State
			END_IF

			fHermesAddOneMsgSend(ADR(a_eMsgSend) , ADR(udiMsgSendBffr) , HermesMsgTypeNotification);

			tyNotificationSnd.tyAvl.bSeverity			:= TRUE;
			tyNotificationSnd.tyAvl.bNotificationCode	:= TRUE;
			tyNotificationSnd.tyAvl.bDescription		:= TRUE;
			tyNotificationSnd.tyData.eSeverity			:= HermesSeverityFatalError;
			tyNotificationSnd.tyData.iNotificationCode	:= UDINT_TO_INT(udiStatus2);
			tyNotificationSnd.tyData.sDescription		:= a_tyAlmText[udiStatus2].sAlmText;

		END_IF

	END_IF

END_ACTION
```

#### Act_Background_ChkParamRcv.st - Do Not Change!!!
```iecst
(** 2019-03-25 **)
ACTION Act_Background_ChkParamRcv:

	IF eStatus2 <> Error THEN

		//Check Parameter Receive
		IF tyMsgTypeRcv.bServiceDescription = TRUE THEN
			udiStatus2	:= fHermesChkParamSD(tyServiceDescriptionRcv , p_tyParam.iLaneID);

			IF udiStatus2 = 2731 THEN
				udiStatus2	:= 0;
			END_IF

			IF udiStatus2 <> 0 THEN
				eStatus2	:= Error;

				IF udiStatus2 = 2726 THEN
					udiStatus2	:= 10086;	//LaneId Mismatch While Checking Service Description
				ELSIF udiStatus2 = 2727 THEN
					udiStatus2	:= 10087;	//MachineId Missing While Checking Service Description
				ELSIF udiStatus2 = 2728 THEN
					udiStatus2	:= 10088;	//LandId Out Of Range While Checking Service Description
				ELSIF udiStatus2 = 2729 THEN
					udiStatus2	:= 10089;	//LandId Missing While Checking Service Description
				ELSIF udiStatus2 = 2730 THEN
					udiStatus2	:= 10090;	//Version Missing While Checking Service Description
				ELSIF udiStatus2 = 2731 THEN
					udiStatus2	:= 10091;	//SupportedFeatures Missing While Checking Service Description
				END_IF

				fHermesAddOneMsgSend(ADR(a_eMsgSend) , ADR(udiMsgSendBffr) , HermesMsgTypeNotification);

				tyNotificationSnd.tyAvl.bSeverity			:= TRUE;
				tyNotificationSnd.tyAvl.bNotificationCode	:= TRUE;
				tyNotificationSnd.tyAvl.bDescription		:= TRUE;
				tyNotificationSnd.tyData.eSeverity			:= HermesSeverityFatalError;
				tyNotificationSnd.tyData.iNotificationCode	:= UDINT_TO_INT(udiStatus2);
				tyNotificationSnd.tyData.sDescription		:= a_tyAlmText[udiStatus2].sAlmText;

			END_IF
		END_IF

		IF tyMsgTypeRcv.bNotification = TRUE THEN
			udiStatus2	:= fHermesChkParamN(tyNotificationRcv);

			IF udiStatus2 <> 0 THEN
				eStatus2	:= Error;

				IF udiStatus2 = 2732 THEN
					udiStatus2	:= 10092;	//NotificationCode Out Of Range While Checking Notification
				ELSIF udiStatus2 = 2733 THEN
					udiStatus2	:= 10093;	//NotificationCode Missing While Checking Notification
				ELSIF udiStatus2 = 2734 THEN
					udiStatus2	:= 10094;	//Severity Missing While Checking Notification
				ELSIF udiStatus2 = 2735 THEN
					udiStatus2	:= 10095;	//Description Missing While Checking Notification
				END_IF

				fHermesAddOneMsgSend(ADR(a_eMsgSend) , ADR(udiMsgSendBffr) , HermesMsgTypeNotification);

				tyNotificationSnd.tyAvl.bSeverity			:= TRUE;
				tyNotificationSnd.tyAvl.bNotificationCode	:= TRUE;
				tyNotificationSnd.tyAvl.bDescription		:= TRUE;
				tyNotificationSnd.tyData.eSeverity			:= HermesSeverityFatalError;
				tyNotificationSnd.tyData.iNotificationCode	:= UDINT_TO_INT(udiStatus2);
				tyNotificationSnd.tyData.sDescription		:= a_tyAlmText[udiStatus2].sAlmText;

			END_IF
		END_IF

		IF tyMsgTypeRcv.bBoardAvailable = TRUE THEN
			udiStatus2	:= fHermesChkParamBA(tyBoardAvailableRcv);

			IF udiStatus2 <> 0 THEN
				eStatus2	:= Error;

				IF udiStatus2 = 2736 THEN
					udiStatus2	:= 10096;	//BoardId Missing While Checking Board Available
				ELSIF udiStatus2 = 2737 THEN
					udiStatus2	:= 10097;	//BoardIdCreatedBy Missing While Checking Board Available
				ELSIF udiStatus2 = 2738 THEN
					udiStatus2	:= 10098;	//FailedBoard Missing While Checking Board Available
				ELSIF udiStatus2 = 2739 THEN
					udiStatus2	:= 10099;	//FlippedBoard Missing While Checking Board Available
				END_IF

				fHermesAddOneMsgSend(ADR(a_eMsgSend) , ADR(udiMsgSendBffr) , HermesMsgTypeNotification);

				tyNotificationSnd.tyAvl.bSeverity			:= TRUE;
				tyNotificationSnd.tyAvl.bNotificationCode	:= TRUE;
				tyNotificationSnd.tyAvl.bDescription		:= TRUE;
				tyNotificationSnd.tyData.eSeverity			:= HermesSeverityError;
				tyNotificationSnd.tyData.iNotificationCode	:= UDINT_TO_INT(udiStatus2);
				tyNotificationSnd.tyData.sDescription		:= a_tyAlmText[udiStatus2].sAlmText;

			END_IF
		END_IF

		IF tyMsgTypeRcv.bTransportFinished = TRUE THEN
			udiStatus2	:= fHermesChkParamTF(tyTransportFinished);

			IF udiStatus2 <> 0 THEN
				eStatus2	:= Error;

				IF udiStatus2 = 2744 THEN
					udiStatus2	:= 10100;	//TransferState Missing While Checking Transport Finished
				ELSIF udiStatus2 = 2745 THEN
					udiStatus2	:= 10101;	//BoardId Missing While Checking Transport Finished
				END_IF

				fHermesAddOneMsgSend(ADR(a_eMsgSend) , ADR(udiMsgSendBffr) , HermesMsgTypeNotification);

				tyNotificationSnd.tyAvl.bSeverity			:= TRUE;
				tyNotificationSnd.tyAvl.bNotificationCode	:= TRUE;
				tyNotificationSnd.tyAvl.bDescription		:= TRUE;
				tyNotificationSnd.tyData.eSeverity			:= HermesSeverityError;
				tyNotificationSnd.tyData.iNotificationCode	:= UDINT_TO_INT(udiStatus2);
				tyNotificationSnd.tyData.sDescription		:= a_tyAlmText[udiStatus2].sAlmText;

			END_IF
		END_IF

		IF tyMsgTypeRcv.bBoardForecast = TRUE THEN
			IF bFeatureBoardForecast = TRUE THEN

				udiStatus2	:= fHermesChkParamBF(tyBoardForecastRcv);

				IF udiStatus2 <> 0 THEN
					eStatus2	:= Error;

					IF udiStatus2 = 2764 THEN
						udiStatus2	:= 10102;	//FailedBoard Missing While Checking Board Forecast

					ELSIF udiStatus2 = 2765 THEN
						udiStatus2	:= 10103;	//FlippedBoard Missing While Checking Board Forecast
					END_IF

					fHermesAddOneMsgSend(ADR(a_eMsgSend) , ADR(udiMsgSendBffr) , HermesMsgTypeNotification);

					tyNotificationSnd.tyAvl.bSeverity			:= TRUE;
					tyNotificationSnd.tyAvl.bNotificationCode	:= TRUE;
					tyNotificationSnd.tyAvl.bDescription		:= TRUE;
					tyNotificationSnd.tyData.eSeverity			:= HermesSeverityError;
					tyNotificationSnd.tyData.iNotificationCode	:= UDINT_TO_INT(udiStatus2);
					tyNotificationSnd.tyData.sDescription		:= a_tyAlmText[udiStatus2].sAlmText;

				END_IF

			ELSE
				tyMsgTypeRcv.bBoardForecast := FALSE;
			END_IF
		END_IF

		IF tyMsgTypeRcv.bCommand = TRUE THEN
			udiStatus2 := fHermesChkParamCommand(tyCommandRcv);

			IF udiStatus2 <> 0 THEN
				eStatus2	:= Error;

//				IF udiStatus2 = 2764 THEN
//					udiStatus2	:= 10102;	//FailedBoard Missing While Checking Board Forecast
//
//				ELSIF udiStatus2 = 2765 THEN
//					udiStatus2	:= 10103;	//FlippedBoard Missing While Checking Board Forecast
//				END_IF

				fHermesAddOneMsgSend(ADR(a_eMsgSend) , ADR(udiMsgSendBffr) , HermesMsgTypeNotification);

				tyNotificationSnd.tyAvl.bSeverity			:= TRUE;
				tyNotificationSnd.tyAvl.bNotificationCode	:= TRUE;
				tyNotificationSnd.tyAvl.bDescription		:= TRUE;
				tyNotificationSnd.tyData.eSeverity			:= HermesSeverityError;
				tyNotificationSnd.tyData.iNotificationCode	:= UDINT_TO_INT(udiStatus2);
				tyNotificationSnd.tyData.sDescription		:= a_tyAlmText[udiStatus2].sAlmText;

			END_IF

		END_IF

	END_IF

END_ACTION
```

#### Act_Background_Sequence.st - Do Not Change!!!
```iecst
 (** 2019-05-04 **)
ACTION Act_Background_Sequence:

	IF eStatus1 <> Error THEN

		IF p_bOpsRun = FALSE THEN
			p_bRcvIncompl	:= TRUE;
		END_IF

		IF tyMsgTypeRcv.bTransportFinished = TRUE THEN
			IF tyTransportFinished.tyData.eTransferState = HermesTransferStateNotStarted THEN
				p_bRcvNotStart	:= TRUE;
			ELSIF tyTransportFinished.tyData.eTransferState = HermesTransferStateIncomplete THEN
				p_bRcvIncompl	:= TRUE;
			END_IF
		END_IF

		bBlkUS := bBABlkUS OR  bBFBlkUS OR bManuallInsertLastZone
			OR bReverseDSSndBfWBrdID
			OR bReverseRcvBlkUS
			OR p_bHermesSwitchtoRvrseTransport;

		bBoardAvailableRcved := tyMsgTypeRcv.bBoardAvailable;

		//Sequence
		fbSequenceUS.bRstState		:= bRstState;
		fbSequenceUS.bRdyRcv		:= (p_bRdyRcv) AND (eStatus2 <> Error);
		fbSequenceUS.bBlkUS			:= bBlkUS;
		fbSequenceUS.bRdyTransport	:= p_bRdyTransport;
		fbSequenceUS.bRcvCompl		:= p_bRcvCompl;
		fbSequenceUS.bRcvIncompl	:= p_bRcvIncompl;
		fbSequenceUS.bRcvNotStart	:= p_bRcvNotStart;
		fbSequenceUS.bProcessBoardForecastId     	:= bProcessBoardForecastId; //Received BoardForecastId

		fbSequenceUS(bEn := TRUE);

		bNotAvlNotRdy                               := fbSequenceUS.bNotAvlNotRdy;

		bUSRdy		                               	:= fbSequenceUS.bUSRdy; //bUSRdy:= (eState = HermesStateBoardAvailable) OR (eState = HermesStateAvailableAndReady) OR (eState >= HermesStateTransporting);
		bDSRdy		                               	:= fbSequenceUS.bDSRdy;
		bTransporting                             	:= fbSequenceUS.bTransporting;
		bStopTransport                            	:= fbSequenceUS.bStopTransport;
		bUSGdRdy                                   	:= (tyBoardAvailableRcv.tyAvl.bFailedBoard = FALSE) OR ((tyBoardAvailableRcv.tyAvl.bFailedBoard = TRUE) AND (tyBoardAvailableRcv.tyData.eFailedBoard <> HermesFailedBoard));
		bDSGdRdy                                   	:= (tyMachineReady.tyAvl.bFailedBoard = FALSE) OR ((tyMachineReady.tyAvl.bFailedBoard = TRUE) AND (tyMachineReady.tyData.eFailedBoard <> HermesFailedBoard));

		//Action (defined 1 as bypass, 2 as flip)
		iAction										:= (tyBoardAvailableRcv.tyAvl.bAction = TRUE)*(tyBoardAvailableRcv.tyData.iAction);

		IF fbSequenceUS.eState >= HermesStateNotAvailableNotReady THEN
			bHandshakeDone	:= TRUE;
		ELSE
			bHandshakeDone	:= FALSE;
		END_IF

		IF EDGEPOS(fbSequenceUS.eState = HermesStateTransporting) THEN
			p_bRcvCompl		:= FALSE;
			p_bRcvIncompl	:= FALSE;
			p_bRcvNotStart	:= FALSE;
		END_IF

		IF fbSequenceUS.eMsgTypeSnd = HermesMsgTypeServiceDescription THEN
			fHermesAddOneMsgSend(ADR(a_eMsgSend) , ADR(udiMsgSendBffr) , HermesMsgTypeServiceDescription);

			tyServiceDescriptionSnd.tyData.sMachineId                                       := p_sMcId;
			tyServiceDescriptionSnd.tyData.iLaneId											:= p_tyParam.iLaneID;
			tyServiceDescriptionSnd.tyData.sInterfaceId										:= p_tyParam.sUpstreamInterfaceId;
			tyServiceDescriptionSnd.tyData.sVersion											:= p_sVersion;
			tyServiceDescriptionSnd.tyData.tySupportedFeatures.bFeatureCheckAliveResponse	:= (p_tyParam.bFeatureCheckAliveResponse) AND (p_tyParam.tRcvAlive <> T#0s) AND (p_tyParam.tSndAlive <> T#0s);
			tyServiceDescriptionSnd.tyData.tySupportedFeatures.bFeatureBoardForecast		:= p_tyParam.bFeatureBoardForecast;
			tyServiceDescriptionSnd.tyData.tySupportedFeatures.bFeatureQueryBoardInfo		:= p_tyParam.bFeatureQueryBoardInfo;
			tyServiceDescriptionSnd.tyData.tySupportedFeatures.bFeatureSendBoardInfo		:= FALSE;

			tyServiceDescriptionSnd.tyAvl.bMachineId										:= TRUE;
			tyServiceDescriptionSnd.tyAvl.bLaneId											:= tyServiceDescriptionSnd.tyData.iLaneId <> 0;
			tyServiceDescriptionSnd.tyAvl.bInterfaceId										:= tyServiceDescriptionSnd.tyData.sInterfaceId <> '';
			tyServiceDescriptionSnd.tyAvl.bVersion											:= TRUE;
			tyServiceDescriptionSnd.tyAvl.bSupportedFeatures								:= p_tyParam.bFeatureCheckAliveResponse OR p_tyParam.bFeatureBoardForecast OR p_tyParam.bFeatureQueryBoardInfo;
			tyServiceDescriptionSnd.tyAvl.tySupportedFeatures.bFeatureCheckAliveResponse	:= (p_tyParam.bFeatureCheckAliveResponse) AND (p_tyParam.tRcvAlive <> T#0s) AND (p_tyParam.tSndAlive <> T#0s);
			tyServiceDescriptionSnd.tyAvl.tySupportedFeatures.bFeatureBoardForecast			:= p_tyParam.bFeatureBoardForecast;
			tyServiceDescriptionSnd.tyAvl.tySupportedFeatures.bFeatureQueryBoardInfo		:= p_tyParam.bFeatureQueryBoardInfo;
			tyServiceDescriptionSnd.tyAvl.tySupportedFeatures.bFeatureSendBoardInfo			:= FALSE;

		ELSIF fbSequenceUS.eMsgTypeSnd = HermesMsgTypeMachineReady THEN
			IF bReplyMcRdyId = FALSE THEN

			    fHermesAddOneMsgSend(ADR(a_eMsgSend) , ADR(udiMsgSendBffr) , HermesMsgTypeMachineReady);

		    	tyMachineReady.tyData.eFailedBoard			:= p_eFailedBoard;
				tyMachineReady.tyAvl.bFailedBoard			:= TRUE;
			    tyMachineReady.tyAvl.bForecastId			:= FALSE;
				tyMachineReady.tyAvl.bBoardId				:= FALSE;
			    tyMachineReady.tyAvl.bProductTypeId			:= FALSE;
			    tyMachineReady.tyAvl.bFlippedBoard			:= FALSE;
			    tyMachineReady.tyAvl.bLength				:= FALSE;
			    tyMachineReady.tyAvl.bWidth					:= FALSE;
			    tyMachineReady.tyAvl.bThickness				:= FALSE;
			    tyMachineReady.tyAvl.bConveyorSpeed			:= FALSE;
			    tyMachineReady.tyAvl.bTopClearanceHeight	:= FALSE;
			    tyMachineReady.tyAvl.bBottomClearanceHeight	:= FALSE;
		    	tyMachineReady.tyAvl.bWeight				:= FALSE;
				tyMachineReady.tyAvl.bWorkOrderId			:= FALSE;
				tyMachineReady.tyAvl.bBatchId    			:= FALSE;

			ELSE
				fHermesAddOneMsgSend(ADR(a_eMsgSend) , ADR(udiMsgSendBffr) , HermesMsgTypeMachineReady);

				tyMachineReady.tyData.eFailedBoard			:= p_eFailedBoard;
				tyMachineReady.tyData.sForecastId	        := tyBoardForecastAcc.tyData.sForecastId;
				tyMachineReady.tyData.sProductTypeId	    := p_sRecipeNm;
				tyMachineReady.tyData.rWidth	            := DINT_TO_REAL(p_diWidthInUM) / 1000;
				tyMachineReady.tyAvl.bFailedBoard			:= TRUE;
				tyMachineReady.tyAvl.bForecastId			:= tyBoardForecastAcc.tyData.sForecastId<>'';
				tyMachineReady.tyAvl.bBoardId				:= FALSE;
				tyMachineReady.tyAvl.bProductTypeId			:= tyBoardForecastAcc.tyData.sProductTypeId<>'';
				tyMachineReady.tyAvl.bFlippedBoard			:= FALSE;
				tyMachineReady.tyAvl.bLength				:= FALSE;
				tyMachineReady.tyAvl.bWidth					:= tyMachineReady.tyData.rWidth<>0;
				tyMachineReady.tyAvl.bThickness				:= FALSE;
				tyMachineReady.tyAvl.bConveyorSpeed			:= FALSE;
				tyMachineReady.tyAvl.bTopClearanceHeight	:= FALSE;
				tyMachineReady.tyAvl.bBottomClearanceHeight	:= FALSE;
				tyMachineReady.tyAvl.bWeight				:= FALSE;
				tyMachineReady.tyAvl.bWorkOrderId			:= FALSE;
				tyMachineReady.tyAvl.bBatchId		    	:= FALSE;

			END_IF

		ELSIF fbSequenceUS.eMsgTypeSnd = HermesMsgTypeRevokeMachineReady THEN
			fHermesAddOneMsgSend(ADR(a_eMsgSend) , ADR(udiMsgSendBffr) , HermesMsgTypeRevokeMachineReady);

		ELSIF fbSequenceUS.eMsgTypeSnd = HermesMsgTypeStartTransport THEN
			fHermesAddOneMsgSend(ADR(a_eMsgSend) , ADR(udiMsgSendBffr) , HermesMsgTypeStartTransport);

			tyStartTransport.tyData.sBoardId		:= tyBoardAvailableRcv.tyData.sBoardId;

			tyStartTransport.tyAvl.bBoardId			:= TRUE;
			tyStartTransport.tyAvl.bConveyorSpeed	:= FALSE;

		ELSIF fbSequenceUS.eMsgTypeSnd = HermesMsgTypeStopTransport THEN
			fHermesAddOneMsgSend(ADR(a_eMsgSend) , ADR(udiMsgSendBffr) , HermesMsgTypeStopTransport);

			IF p_bRcvCompl = TRUE THEN
				tyStopTransport.tyData.eTransferState	:= HermesTransferStateComplete;
			ELSIF p_bRcvIncompl = TRUE THEN
				tyStopTransport.tyData.eTransferState	:= HermesTransferStateIncomplete;
			ELSE
				tyStopTransport.tyData.eTransferState	:= HermesTransferStateNotStarted;
			END_IF
			tyStopTransport.tyData.sBoardId				:= tyStartTransport.tyData.sBoardId;

			tyStopTransport.tyAvl.bTransferState		:= TRUE;
			tyStopTransport.tyAvl.bBoardId				:= TRUE;

		END_IF

	END_IF

	bStopTransportSent := fbSequenceUS.eMsgTypeSnd = HermesMsgTypeStopTransport;

END_ACTION
```

#### Act_Background_SequenceTO.st - Do Not Change!!!
```iecst
(** 2019-03-25 **)
ACTION Act_Background_SequenceTO:

	IF (eStatus1 <> Error) AND (eStatus2 <> Error) THEN

		//Time Out
		fbSequenceTO.eState				:= fbSequenceUS.eState;
		fbSequenceTO.tConnTimeOut		:= p_tConnTimeOut;
		fbSequenceTO.tTransportTimeOut	:= DINT_TO_TIME(p_diTransferInTO);
		fbSequenceTO(bEn := TRUE);

		IF fbSequenceTO.udiStatus > 0 AND fbSequenceTO.udiStatus < 65534 THEN

			IF fbSequenceTO.udiStatus = 2912 THEN
				eStatus1	:= Error;
				udiStatus1	:= 10106;	//Service Description Interchange Time Out

				fHermesAddOneMsgSend(ADR(a_eMsgSend) , ADR(udiMsgSendBffr) , HermesMsgTypeNotification);

				tyNotificationSnd.tyAvl.bSeverity			:= TRUE;
				tyNotificationSnd.tyAvl.bNotificationCode	:= TRUE;
				tyNotificationSnd.tyAvl.bDescription		:= TRUE;
				tyNotificationSnd.tyData.eSeverity			:= HermesSeverityFatalError;
				tyNotificationSnd.tyData.iNotificationCode	:= UDINT_TO_INT(udiStatus1);
				tyNotificationSnd.tyData.sDescription		:= a_tyAlmText[udiStatus1].sAlmText;

			ELSIF fbSequenceTO.udiStatus = 2913 THEN
				p_bRcvIncompl	:= TRUE;

				eStatus2	:= Error;
				udiStatus2	:= 10107;	//Transport Time Out

				fHermesAddOneMsgSend(ADR(a_eMsgSend) , ADR(udiMsgSendBffr) , HermesMsgTypeNotification);

				tyNotificationSnd.tyAvl.bSeverity			:= TRUE;
				tyNotificationSnd.tyAvl.bNotificationCode	:= TRUE;
				tyNotificationSnd.tyAvl.bDescription		:= TRUE;
				tyNotificationSnd.tyData.eSeverity			:= HermesSeverityError;
				tyNotificationSnd.tyData.iNotificationCode	:= UDINT_TO_INT(udiStatus2);
				tyNotificationSnd.tyData.sDescription		:= a_tyAlmText[udiStatus2].sAlmText;

			ELSE
				eStatus2	:= Error;
				udiStatus2	:= fbSequenceTO.udiStatus;

				fHermesAddOneMsgSend(ADR(a_eMsgSend) , ADR(udiMsgSendBffr) , HermesMsgTypeNotification);

				tyNotificationSnd.tyAvl.bSeverity			:= TRUE;
				tyNotificationSnd.tyAvl.bNotificationCode	:= TRUE;
				tyNotificationSnd.tyAvl.bDescription		:= TRUE;
				tyNotificationSnd.tyData.eSeverity			:= HermesSeverityFatalError;
				tyNotificationSnd.tyData.iNotificationCode	:= UDINT_TO_INT(udiStatus2);
				tyNotificationSnd.tyData.sDescription		:= a_tyAlmText[udiStatus2].sAlmText;

			END_IF

		END_IF

	END_IF

END_ACTION
```

#### Act_Background_BoardForecast.st - Do Not Change!!!
```iecst
(** 2023-08-01 **)
ACTION Act_Background_BoardForecast:

	//Process BoardForecast(Id) or BoardForecast()
	bFeatureBoardForecast := (p_tyParam.bFeatureBoardForecast = TRUE) AND (tyServiceDescriptionRcv.tyAvl.tySupportedFeatures.bFeatureBoardForecast = TRUE);

	IF bFeatureBoardForecast THEN //if board forecast check message receive
		bBrdForecastRcv := tyMsgTypeRcv.bBoardForecast;

		IF tyMsgTypeRcv.bBoardForecast AND tyBoardForecastRcv.tyData.sForecastId <> '' AND bProcessBoardForecastId = FALSE  AND bBFAccDataReq = FALSE AND bManuallInsertLastZone = FALSE THEN
			bProcessBoardForecastId := TRUE; //Process BoardForecast(Id)
			tyBoardForecastAcc := tyBoardForecastRcv; //capture to process that particular BF
			tyMsgTypeRcv.bBoardForecast := FALSE;

		ELSIF tyMsgTypeRcv.bBoardForecast AND tyBoardForecastRcv.tyData.sForecastId = '' AND bProcessBoardForecastId = FALSE THEN //Process BoardForecast()
			tyBoardForecastAcc := tyBoardForecastRcv;
			tyMsgTypeRcv.bBoardForecast := FALSE;
		END_IF
	ELSE
		bProcessBoardForecastId := FALSE;
	END_IF

	//BF Check
//	IF eStatus2 <> Error THEN
//
//		IF bProcessBoardForecastId AND bNotAvlNotRdy AND (bTransporting = FALSE) AND (p_bOpsRun = TRUE) THEN
//
//			bBFAccDataReq		:= FALSE;
//			bBFBlkUS			:= FALSE;
//			bBFOverWriteSlt  	:= FALSE;
//			bBFOverWriteWidth	:= FALSE;
//
//			IF p_tyParam.bCmpTypeId = TRUE THEN	//"Compare Type ID" Ticked
//
//				IF tyBoardForecastAcc.tyAvl.bProductTypeId = TRUE THEN	//Check if there is Product Type Id in B.F msg
//
//					IF tyBoardForecastAcc.tyData.sProductTypeId <> p_sRecipeNm THEN	//Product Type Id Different
//
//						bBFAccDataReq	:= TRUE;	//Require To Load New Recipe
//						bBFBlkUS		:= TRUE;
//
//						sReqRecipeNm	:= tyBoardForecastAcc.tyData.sProductTypeId;
//						diReqWidthInUM	:= REAL_TO_DINT(tyBoardForecastAcc.tyData.rWidth * 1000);
//
//					ELSE	//Product Type Id Same (After accepted or Originally same)
//
//						IF p_tyParam.bCmpParam = TRUE THEN	//"Compare Param" Ticked
//							IF tyBoardForecastAcc.tyAvl.bThickness AND tyBoardForecastAcc.tyAvl.bTopClearanceHeight AND tyBoardForecastAcc.tyAvl.bBottomClearanceHeight AND p_bBFSltEn THEN	//Camparing Slot Parameters if p_bBFSltEn = TRUE
//								udiStatus2	:= fHermesCmpSlt(tyBoardForecastAcc.tyData.eFlippedBoard , tyBoardForecastAcc.tyData.rThickness , tyBoardForecastAcc.tyData.rTopClearanceHeight , tyBoardForecastAcc.tyData.rBottomClearanceHeight , p_diMinSltValue , p_diMaxSltValue , p_diPitch , p_diSltToSltInUM , p_diTtlSlt);
//
//								IF udiStatus2 <> 0 THEN
//
//									bBFBlkUS		:= TRUE;
//									bProcessBoardForecastId := FALSE;//add
//									eStatus2	:= Error;
//
//									IF udiStatus2 = 2914 THEN
//										udiStatus2	:= 10108;	//Input First Slot Is Invalid
//									ELSIF udiStatus2 = 2915 THEN
//										udiStatus2	:= 10109;	//Input Last Slot Is Invalid
//									ELSIF udiStatus2 = 2916 THEN
//										udiStatus2	:= 10110;	//Input Pitch Is Invalid
//									ELSIF udiStatus2 = 2917 THEN
//										udiStatus2	:= 10111;	//Input Slot To Slot Distance Is Invalid
//									ELSIF udiStatus2 = 2918 THEN
//										udiStatus2	:= 10112;	//Input Total Slot Is Invalid
//									ELSIF udiStatus2 = 2919 THEN
//										udiStatus2	:= 10113;	//Input Thickness Is Invalid
//									ELSIF udiStatus2 = 2920 THEN
//										udiStatus2	:= 10114;	//Input Top Clearance Height Is Invalid
//									ELSIF udiStatus2 = 2921 THEN
//										udiStatus2	:= 10115;	//Input Bottom Clearance Height Is Invalid
//									ELSIF udiStatus2 = 2922 THEN
//										udiStatus2	:= 10116;	//Recipe First Slot Value & Board Available Data Not Match With Same Product Type Id
//									ELSIF udiStatus2 = 2923 THEN
//										udiStatus2	:= 10117;	//Recipe Last Slot Value & Board Available Data Not Match With Same Product Type Id
//									ELSIF udiStatus2 = 2924 THEN
//										udiStatus2	:= 10118;	//Recipe Pitch Value & Board Available Data Not Match With Same Product Type Id
//									END_IF
//
//									fHermesAddOneMsgSend(ADR(a_eMsgSend) , ADR(udiMsgSendBffr) , HermesMsgTypeNotification);
//
//									tyNotificationSnd.tyAvl.bSeverity			:= TRUE;
//									tyNotificationSnd.tyAvl.bNotificationCode	:= TRUE;
//									tyNotificationSnd.tyAvl.bDescription		:= TRUE;
//									tyNotificationSnd.tyData.eSeverity			:= HermesSeverityError;
//									tyNotificationSnd.tyData.iNotificationCode	:= 6; //BoardForecast Error
//									tyNotificationSnd.tyData.sDescription		:= a_tyAlmText[udiStatus2].sAlmText;
//
//								END_IF
//							END_IF
//
//							IF tyBoardForecastAcc.tyAvl.bWidth AND p_bBFWidthEn THEN	//Comparing Width Parameter if p_bBFWidthEn = TRUE
//								IF REAL_TO_DINT(tyBoardForecastAcc.tyData.rWidth * 1000) <> p_diWidthInUM THEN
//
//									bBFBlkUS	:= TRUE;
//									bProcessBoardForecastId := FALSE;//add
//									eStatus2	:= Error;
//									udiStatus2	:= 10119;	//Width Different With Same Product Type Id
//
//									fHermesAddOneMsgSend(ADR(a_eMsgSend) , ADR(udiMsgSendBffr) , HermesMsgTypeNotification);
//
//									tyNotificationSnd.tyAvl.bSeverity			:= TRUE;
//									tyNotificationSnd.tyAvl.bNotificationCode	:= TRUE;
//									tyNotificationSnd.tyAvl.bDescription		:= TRUE;
//									tyNotificationSnd.tyData.eSeverity			:= HermesSeverityError;
//									tyNotificationSnd.tyData.iNotificationCode	:= 6; //BoardForecast Error
//									tyNotificationSnd.tyData.sDescription		:= a_tyAlmText[udiStatus2].sAlmText;
//								ELSE
//									bReplyMcRdyId           := TRUE; //add
//									bProcessBoardForecastId := FALSE; //add
//								END_IF
//							END_IF
//
//						END_IF
//
//					END_IF
//
//				ELSE
//
//					eStatus2	:= Error;
//					udiStatus2	:= 10158;	//Product Type Id Not Receive From Upstream
//					bProcessBoardForecastId := FALSE;//add
//
//					fHermesAddOneMsgSend(ADR(a_eMsgSend) , ADR(udiMsgSendBffr) , HermesMsgTypeNotification);
//
//					tyNotificationSnd.tyAvl.bSeverity			:= TRUE;
//					tyNotificationSnd.tyAvl.bNotificationCode	:= TRUE;
//					tyNotificationSnd.tyAvl.bDescription		:= TRUE;
//					tyNotificationSnd.tyData.eSeverity			:= HermesSeverityError;
//					tyNotificationSnd.tyData.iNotificationCode	:= 6; //BoardForecast Error
//					tyNotificationSnd.tyData.sDescription		:= a_tyAlmText[udiStatus2].sAlmText;
//
//				END_IF
//
//			ELSE	//"Compare Type ID" Not Ticked
//
//				IF p_tyParam.bOverwrite THEN	//"Overwrite" Ticked
//
//					IF tyBoardForecastAcc.tyAvl.bThickness AND tyBoardForecastAcc.tyAvl.bTopClearanceHeight AND tyBoardForecastAcc.tyAvl.bBottomClearanceHeight AND p_bBFSltEn THEN	//Camparing Slot Parameters
//
//						udiStatus2	:= fHermesCmpSlt(tyBoardForecastAcc.tyData.eFlippedBoard , tyBoardForecastAcc.tyData.rThickness , tyBoardForecastAcc.tyData.rTopClearanceHeight , tyBoardForecastAcc.tyData.rBottomClearanceHeight , p_diMinSltValue , p_diMaxSltValue , p_diPitch , p_diSltToSltInUM , p_diTtlSlt);
//
//						IF udiStatus2 <> 0 THEN
//
//							bBFAccDataReq		:= TRUE;
//							bBFBlkUS			:= TRUE;
//							bBFOverWriteSlt	    := TRUE;
//
//							fbGetSlt.eFlippedBrd				:= tyBoardForecastAcc.tyData.eFlippedBoard;
//							fbGetSlt.rThicknessInMM				:= tyBoardForecastAcc.tyData.rThickness;
//							fbGetSlt.rTopClearanceHeightInMM	:= tyBoardForecastAcc.tyData.rTopClearanceHeight;
//							fbGetSlt.rBtmClearanceHeightInMM	:= tyBoardForecastAcc.tyData.rBottomClearanceHeight;
//							fbGetSlt.diSltToSltInUM				:= p_diSltToSltInUM;
//							fbGetSlt.diTtlSlt					:= p_diTtlSlt;
//							fbGetSlt;
//
//							diReqMinSltValue	:= fbGetSlt.diMinSltValue;
//							diReqMaxSltValue	:= fbGetSlt.diMaxSltValue;
//							diReqPitch			:= fbGetSlt.diPitch;
//
//						END_IF
//
//					END_IF
//
//					IF tyBoardForecastAcc.tyAvl.bWidth AND p_bBFWidthEn THEN	//Comparing Width Parameter
//						IF REAL_TO_DINT(tyBoardForecastAcc.tyData.rWidth * 1000) <> p_diWidthInUM THEN
//
//							bBFAccDataReq		:= TRUE;
//							bBFBlkUS			:= TRUE;
//							bBFOverWriteWidth	:= TRUE;
//
//							diReqWidthInUM	:= REAL_TO_DINT(tyBoardForecastAcc.tyData.rWidth * 1000);
//						ELSE
//							bReplyMcRdyId           := TRUE; //add
//							bProcessBoardForecastId := FALSE; //add
//						END_IF
//					END_IF
//
//				ELSE	//"Compare Type ID" Not Ticked and "Overwrite" Not Ticked, Error if not same
//
//					IF tyBoardForecastAcc.tyAvl.bThickness AND tyBoardForecastAcc.tyAvl.bTopClearanceHeight AND tyBoardForecastAcc.tyAvl.bBottomClearanceHeight AND p_bBFSltEn AND p_bRdyRcv THEN	//Camparing Slot Parameters
//						udiStatus2	:= fHermesCmpSlt(tyBoardForecastAcc.tyData.eFlippedBoard , tyBoardForecastAcc.tyData.rThickness , tyBoardForecastAcc.tyData.rTopClearanceHeight , tyBoardForecastAcc.tyData.rBottomClearanceHeight , p_diMinSltValue , p_diMaxSltValue , p_diPitch , p_diSltToSltInUM , p_diTtlSlt);
//
//						IF udiStatus2 <> 0 THEN
//
//							bBFBlkUS		:= TRUE;
//							bProcessBoardForecastId := FALSE;//add
//							eStatus2	:= Error;
//
//							IF udiStatus2 = 2914 THEN
//								udiStatus2	:= 10120;	//Input First Slot Is Invalid
//							ELSIF udiStatus2 = 2915 THEN
//								udiStatus2	:= 10121;	//Input Last Slot Is Invalid
//							ELSIF udiStatus2 = 2916 THEN
//								udiStatus2	:= 10122;	//Input Pitch Is Invalid
//							ELSIF udiStatus2 = 2917 THEN
//								udiStatus2	:= 10123;	//Input Slot To Slot Distance Is Invalid
//							ELSIF udiStatus2 = 2918 THEN
//								udiStatus2	:= 10124;	//Input Total Slot Is Invalid
//							ELSIF udiStatus2 = 2919 THEN
//								udiStatus2	:= 10125;	//Input Thickness Is Invalid
//							ELSIF udiStatus2 = 2920 THEN
//								udiStatus2	:= 10126;	//Input Top Clearance Height Is Invalid
//							ELSIF udiStatus2 = 2921 THEN
//								udiStatus2	:= 10127;	//Input Bottom Clearance Height Is Invalid
//							ELSIF udiStatus2 = 2922 THEN
//								udiStatus2	:= 10128;	//Recipe First Slot Value & Board Available Data Not Match With Same Product Type Id
//							ELSIF udiStatus2 = 2923 THEN
//								udiStatus2	:= 10129;	//Recipe Last Slot Value & Board Available Data Not Match With Same Product Type Id
//							ELSIF udiStatus2 = 2924 THEN
//								udiStatus2	:= 10130;	//Recipe Pitch Value & Board Available Data Not Match With Same Product Type Id
//							END_IF
//
//							fHermesAddOneMsgSend(ADR(a_eMsgSend) , ADR(udiMsgSendBffr) , HermesMsgTypeNotification);
//
//							tyNotificationSnd.tyAvl.bSeverity			:= TRUE;
//							tyNotificationSnd.tyAvl.bNotificationCode	:= TRUE;
//							tyNotificationSnd.tyAvl.bDescription		:= TRUE;
//							tyNotificationSnd.tyData.eSeverity			:= HermesSeverityError;
//							tyNotificationSnd.tyData.iNotificationCode	:= 6; //BoardForecast Error
//							tyNotificationSnd.tyData.sDescription		:= a_tyAlmText[udiStatus2].sAlmText;
//
//						END_IF
//					END_IF
//
//					IF tyBoardForecastAcc.tyAvl.bWidth AND p_bBFWidthEn AND p_bRdyRcv THEN	//Comparing Width Parameter
//						IF REAL_TO_DINT(tyBoardForecastAcc.tyData.rWidth * 1000) <> p_diWidthInUM THEN
//
//							bBFBlkUS		:= TRUE;
//							bProcessBoardForecastId := FALSE;//add
//							eStatus2	:= Error;
//							udiStatus2	:= 10131;	//Width Different With Same Product Type Id
//
//							fHermesAddOneMsgSend(ADR(a_eMsgSend) , ADR(udiMsgSendBffr) , HermesMsgTypeNotification);
//
//							tyNotificationSnd.tyAvl.bSeverity			:= TRUE;
//							tyNotificationSnd.tyAvl.bNotificationCode	:= TRUE;
//							tyNotificationSnd.tyAvl.bDescription		:= TRUE;
//							tyNotificationSnd.tyData.eSeverity			:= HermesSeverityError;
//							tyNotificationSnd.tyData.iNotificationCode	:= 6; //BoardForecast Error
//							tyNotificationSnd.tyData.sDescription		:= a_tyAlmText[udiStatus2].sAlmText;
//						ELSE
//							bReplyMcRdyId           := TRUE; //add
//							bProcessBoardForecastId := FALSE; //add
//						END_IF
//					END_IF
//
//				END_IF
//
//			END_IF
//
//
//
//		ELSIF bProcessBoardForecastId = FALSE OR bNotAvlNotRdy =FALSE OR bTransporting = TRUE THEN
//
//			bBFAccDataReq		:= FALSE;
//			bBFBlkUS			:= FALSE;
//			bBFOverWriteSlt	    := FALSE;
//			bBFOverWriteWidth	:= FALSE;
//
//		END_IF
//
//	ELSE
//
//		bBFAccDataReq		:= FALSE;
//		bBFBlkUS			:= TRUE;
//		bBFOverWriteSlt	    := FALSE;
//		bBFOverWriteWidth	:= FALSE;
//
//	END_IF

END_ACTION
```

#### Act_Background_ChkAliveSendPing.st - Do Not Change!!!
```iecst
(** 2019-05-30 **)
ACTION Act_Background_ChkAliveSendPing:

	IF eStatus1 <> Error THEN

		//Check Alive Send Ping
		fbCheckAliveSendPing.bDataRcv		:= tyMsgTypeRcv.bCheckAlivePong;
		fbCheckAliveSendPing.tyDataRcv		:= tyCheckAlivePongRcv;
		fbCheckAliveSendPing.tyDTStructure	:= p_tyDTStructure;
		fbCheckAliveSendPing.tSendTm		:= p_tyParam.tSndAlive;
		fbCheckAliveSendPing.tRcvTimeOut	:= p_tyParam.tRcvAlive;
		fbCheckAliveSendPing(bEn := TRUE);

		IF fbCheckAliveSendPing.udiStatus > 0 AND fbCheckAliveSendPing.udiStatus < 65534 THEN
			eStatus1	:= Error;

			IF fbCheckAliveSendPing.udiStatus = 2768 THEN
				udiStatus1	:= 10133;	//Waiting Check Alive Time Out
			ELSIF fbCheckAliveSendPing.udiStatus = 2769 THEN
				udiStatus1	:= 10134;	//Check Alive Id Mismatch
			ELSE
				udiStatus1	:= fbCheckAliveSendPing.udiStatus;
			END_IF

			fHermesAddOneMsgSend(ADR(a_eMsgSend) , ADR(udiMsgSendBffr) , HermesMsgTypeNotification);

			tyNotificationSnd.tyAvl.bSeverity			:= TRUE;
			tyNotificationSnd.tyAvl.bNotificationCode	:= TRUE;
			tyNotificationSnd.tyAvl.bDescription		:= TRUE;
			tyNotificationSnd.tyData.eSeverity			:= HermesSeverityFatalError;
			tyNotificationSnd.tyData.iNotificationCode	:= UDINT_TO_INT(udiStatus1);
			tyNotificationSnd.tyData.sDescription		:= a_tyAlmText[udiStatus1].sAlmText;

		ELSE
			IF EDGEPOS(fbCheckAliveSendPing.bDataSend) THEN
				fHermesAddOneMsgSend(ADR(a_eMsgSend) , ADR(udiMsgSendBffr) , HermesMsgTypeCheckAlivePing);
				tyCheckAlivePingSnd	:= fbCheckAliveSendPing.tyDataSend;
			END_IF

		END_IF

		tyMsgTypeRcv.bCheckAlivePong	:= FALSE;	//Reset Check Alive Pong

	END_IF

END_ACTION
```

#### Act_Background_ChkAliveRcvPing.st - Do Not Change!!!
```iecst
(** 2019-05-30 **)
ACTION Act_Background_ChkAliveRcvPing:

	IF eStatus1 <> Error THEN

		//Check Alive Receive Ping
		fbCheckAliveRcvPing.bDataRcv	:= tyMsgTypeRcv.bCheckAlivePing;
		fbCheckAliveRcvPing.tyDataRcv	:= tyCheckAlivePingRcv;
		fbCheckAliveRcvPing(bEn := TRUE);

		IF fbCheckAliveRcvPing.udiStatus > 0 AND fbCheckAliveRcvPing.udiStatus < 65534 THEN
			eStatus1	:= Error;
			udiStatus1	:= fbCheckAliveRcvPing.udiStatus;

		ELSE
			IF EDGEPOS(fbCheckAliveRcvPing.bDataSend) THEN
				fHermesAddOneMsgSend(ADR(a_eMsgSend) , ADR(udiMsgSendBffr) , HermesMsgTypeCheckAlivePong);
				tyCheckAlivePongSnd	:= fbCheckAliveRcvPing.tyDataSend;
			END_IF

		END_IF

		tyMsgTypeRcv.bCheckAlivePing	:= FALSE;	//Reset Check Alive Ping

	END_IF

END_ACTION
```

#### Act_Background_Command.st - Do Not Change!!!
```iecst
(** 2021-08-01 **)
ACTION Act_Background_Command:
	//tyServiceDescriptionRcv.tyAvl.tySupportedFeatures.bFeatureCommand = TRUE AND p_tyParam.bFeatureCommand AND

	IF NOT(p_tyParam.bFeatureCommand AND tyServiceDescriptionRcv.tyAvl.tySupportedFeatures.bFeatureCommand AND bHandshakeDone) THEN
		IF tyCommandParam.a_eCommandSndQ[0] <> HermesCommandUndefined THEN
			fHermesRmvOneCmdTyp(ADR(tyCommandParam.a_eCommandSndQ),ADR(tyCommandParam.udiMsgCmdBffr));
		END_IF
	ELSE
		IF eStatus2 <> Error THEN
			//receive command

			IF tyMsgTypeRcv.bCommand THEN
				tyCommandParam.usiCommandIdx :=  tyCommandParam.usiCommandIdx + 1;
				tyCommandParam.eCommand := tyCommandRcv.tyData.eCommand;
				tyMsgTypeRcv.bCommand  := FALSE;
			END_IF

			//sending
			IF  tyCommandParam.a_eCommandSndQ[0] <> HermesCommandUndefined THEN
				//Queuing for sending command
				fHermesAddOneMsgSend(ADR(a_eMsgSend) , ADR(udiMsgSendBffr) , HermesMsgTypeCommand);
				tyCommandSnd.tyData.eCommand :=  tyCommandParam.a_eCommandSndQ[0];
				tyCommandSnd.tyAvl.bCommand :=  TRUE;
				fHermesRmvOneCmdTyp(ADR(tyCommandParam.a_eCommandSndQ),ADR(tyCommandParam.udiMsgCmdBffr));
			END_IF
		END_IF
	END_IF

END_ACTION
```

#### Act_Background_Route.st - Do Not Change!!!
```iecst
(** 2021-08-01 **)
ACTION Act_Background_Route:

	//US Routing function

	//iGotoLane 0 Default Lane
	//iGotoLane 1 Route1
	IF NOT(p_bProcessRouteEn) THEN
		bReverseDSSndBfWBrdID := FALSE;
		bManualRmvBrdCond := FALSE;
		iGotoLane	:= 0;
		bProcessRouteReversal := FALSE;
		bTriggerRouteReversal := FALSE;
	ELSE
		// reversal condition
		IF EDGEPOS(tyBoardAvailableRcv.tyData.iRoute  = 900) THEN //flipping station reversal condition
			bProcessRouteReversal := TRUE;
		ELSIF EDGEPOS(tyBoardAvailableRcv.tyAvl.bFlippedBoard  AND tyBoardAvailableRcv.tyData.eFlippedBoard = HermesFlippedBoardTopSideUp) THEN
			bTriggerRouteReversal := TRUE;
		END_IF

		//receiving Route
		IF	NOT(tyBoardAvailableRcv.tyAvl.bRoute)   THEN
			iGotoLane := 0; //default, depend on priority
		ELSE
			IF  p_bManualRmvRoute AND tyBoardAvailableRcv.tyData.iRoute  = 999  THEN
				bManualRmvBrdCond := TRUE;

			ELSIF p_bReturnRoute AND (
				(bProcessRouteReversal AND bProcessRouteMachine
				OR
				bTriggerRouteReversal AND bTriggerRouteMachine)
				OR bReverseDSSndBfWBrdID) THEN
				IF bProcessRouteReversal  THEN //Route Guide (900),flipper as downstream
					bReverseDSSndBfWBrdID := TRUE;
					bTriggerUpdateRoute  := FALSE;
					bProcessRouteReversal := FALSE;
				ELSIF bTriggerRouteReversal THEN //process as downstream
					bReverseDSSndBfWBrdID := TRUE;
					bTriggerUpdateRoute  := TRUE;
					bTriggerRouteReversal := FALSE;
				END_IF

				//Reset
				fbRstReverseDSSndBF(IN:= bReverseDSSndBfWBrdID AND NOT(p_bReceiveReverseUSMcRdy));
				IF (bReverseDSSndBfWBrdID AND p_bReceiveReverseUSMcRdy) OR fbRstReverseDSSndBF.Q THEN
					bReverseDSSndBfWBrdID := FALSE;
					bTriggerUpdateRoute := FALSE;
				END_IF
			ELSIF p_bNomRouteEn THEN
				iMinDis := 0;
				FOR usidx := 0 TO 2 DO
					//bChecking Closest Route
					IF tyBoardAvailableRcv.tyData.iRoute = pa_tyHermesDSParam[usidx].iLaneID THEN
						iGotoLane := usidx; //iGotoLane switch direction
						EXIT;
					ELSIF iMinDis = 0 THEN
						iMinDis := ABS(tyBoardAvailableRcv.tyData.iRoute - pa_tyHermesDSParam[usidx].iLaneID);
						iGotoLane := usidx;
					ELSE
						IF iMinDis > ABS(tyBoardAvailableRcv.tyData.iRoute - pa_tyHermesDSParam[usidx].iLaneID) THEN
							iGotoLane := usidx;
							iMinDis := ABS(tyBoardAvailableRcv.tyData.iRoute - pa_tyHermesDSParam[usidx].iLaneID);
						END_IF
					END_IF
				END_FOR
			END_IF
		END_IF

		//Process 900
		//when to reset block DS signal

		//Process 999
		//fbRstReverseDSSndBF(IN:= bManualRmvBrdCond);

	//	bBlkUS := bBlkUS OR bReverseDSSndBfWBrdID; //OR p_bSwitchtoReverseReceive;
	END_IF

	//reverse route, input receiving
	IF NOT(p_bReverseReceiveRoute) THEN
		bSwitchtoReverseReceive := FALSE;
	ELSE
		//process Reverse Input
		IF bSwitchtoReverseReceive = FALSE  AND EDGEPOS(p_tyDSHermesCurrBASnd.tyData.sBoardId = tyBoardForecastRcv.tyData.sBoardId AND tyBoardForecastRcv.tyData.sBoardId <> '' ) THEN
			bSwitchtoReverseReceive := TRUE; //when to reset ReverseRcv back , if the BASnd not the same anymore
		ELSIF bSwitchtoReverseReceive = TRUE
			AND (EDGEPOS(tyMsgTypeRcv.bTransportFinished AND tyTransportFinished.tyData.eTransferState = HermesTransferStateComplete )
			OR EDGEPOS(tyMsgTypeRcv.bBoardForecast AND tyBoardForecastRcv.tyData.sBoardId = '' )) THEN
			bSwitchtoReverseReceive := FALSE;
		END_IF
		fbRstReverseRcvGate(IN:= bSwitchtoReverseReceive);
		bNotifyRstReverseRcvGate := fbRstReverseRcvGate.Q;
		//	bBlkUS := bBlkUS OR NOT(bSwitchtoReverseReceive);

		bReverseRcvBlkUS := NOT(bSwitchtoReverseReceive);
	END_IF

	//bBlkUS := bBlkUS OR p_bUSHermes2SwitchtoReverseRcv;
END_ACTION
```

#### Act_Background_NotificationSnd.st - Do Not Change!!!
```iecst
(** 2019-03-15 **)
ACTION Act_Background_NotificationSnd:

	IF a_eMsgSend[0] = HermesMsgTypeNotification THEN
		bRstConnection	:= fHermesNotificationRstConn(tyNotificationSnd) OR bRstConnection; //Fatal Error = Reset Connection, Error no reset
//		bRstState		:= fHermesNotificationRstState(tyNotificationSnd) OR bRstState;
	END_IF

END_ACTION
```

#### Act_Background_QueryBoardInfo.st - Do Not Change!!!
```iecst
(** 2021-08-01 **)
ACTION Act_Background_QueryBoardInfo:
	IF NOT(tyServiceDescriptionRcv.tyAvl.tySupportedFeatures.bFeatureSendBoardInfo = TRUE AND p_tyParam.bFeatureQueryBoardInfo AND bHandshakeDone) THEN
		bRcvBoardInfoOk              := FALSE;;
		bManuallInsertLastZone        := FALSE;
		bRcvBoardInfoIncompl := FALSE;
	ELSE
		IF eStatus2 <> Error THEN

			IF EDGEPOS(p_bQueryBoardInfo) THEN

				fHermesAddOneMsgSend(ADR(a_eMsgSend) , ADR(udiMsgSendBffr) , HermesMsgTypeQueryBoardInfo);

				tyQueryBoardInfo.tyData.sTopBarcode						            := p_sTopBarcode;
				tyQueryBoardInfo.tyData.sBottomBarcode							    := p_sBottomBarcode;

				tyQueryBoardInfo.tyAvl.bTopBarcode									:= tyQueryBoardInfo.tyData.sTopBarcode <> '';
				tyQueryBoardInfo.tyAvl.bBottomBarcode							    := tyQueryBoardInfo.tyData.sBottomBarcode <>'';

			END_IF

			IF tyMsgTypeRcv.bSendBoardInfo THEN

				IF p_bQueryBoardInfo AND (udiStatus2 = 0) THEN //After CmpParamRcv
					IF tySendBoardInfoRcv.tyAvl.bBoardId AND tySendBoardInfoRcv.tyAvl.bBoardIdCreatedBy AND p_bManualInsertZoneHvBrd = FALSE AND p_bManualInsertEndSen = FALSE THEN //Wait Empty

						bRcvBoardInfoOk              := TRUE;
						tySendBoardInfoAcc          := tySendBoardInfoRcv;
						tyMsgTypeRcv.bSendBoardInfo := FALSE;

					ELSIF ((tySendBoardInfoRcv.tyAvl.bBoardId = FALSE) OR (tySendBoardInfoRcv.tyAvl.bBoardIdCreatedBy = FALSE)) THEN //no BoardId or BoardIdCreatedBy
						bRcvBoardInfoIncompl := TRUE;
						bManuallInsertLastZone         := FALSE;
						tyMsgTypeRcv.bSendBoardInfo := FALSE;
					END_IF

				ELSIF p_bQueryBoardInfo = FALSE THEN
					tyMsgTypeRcv.bSendBoardInfo     := FALSE;
				END_IF

			END_IF

			IF 	bRcvBoardInfoOk = TRUE THEN
				bManuallInsertLastZone        := TRUE; //Board data received from upstream, block Upstream to allow manual insert

				tyInfoData1.sProgNm		:= p_sProgNm;
				tyInfoData1.udiCode		:= 10000;
				tyInfoData1.eSeverity	:= AlmSeverityInfo;
				tyInfoData1.sAlmMsg		:= p_sInfoMsg1;

				IF p_bTransportFinished THEN

					bRcvBoardInfoOk := FALSE;
					bManuallInsertLastZone        := FALSE;
				END_IF

			ELSIF bRcvBoardInfoIncompl = TRUE THEN //receive dummy, no need block upstream

				tyInfoData2.sProgNm		:= p_sProgNm;
				tyInfoData2.udiCode		:= 10000;
				tyInfoData2.eSeverity	:= AlmSeverityInfo;
				tyInfoData2.sAlmMsg		:= p_sInfoMsg2;

			END_IF

			IF p_bQueryBoardInfo = FALSE THEN

				//Clear Info Message 1
				tyInfoData1.sProgNm		:= '';
				tyInfoData1.udiCode		:= 0;
				tyInfoData1.eSeverity	:= AlmSeverityNA;
				tyInfoData1.sAlmMsg		:= '';
				bRcvBoardInfoOk := FALSE;
				bManuallInsertLastZone        := FALSE;

				//Clear Info Message 2
				tyInfoData2.sProgNm		:= '';
				tyInfoData2.udiCode		:= 0;
				tyInfoData2.eSeverity	:= AlmSeverityNA;
				tyInfoData2.sAlmMsg		:= '';
				bRcvBoardInfoIncompl := FALSE;

			END_IF

		END_IF

	END_IF

END_ACTION
```

#### Act_Background_TCPSend.st - Do Not Change!!!
```iecst
(** 2019-06-10 **)
ACTION Act_Background_TCPSend:

	//Message Send (Generate XML Message)
	IF a_eMsgSend[0] <> HermesMsgTypeNA THEN

		IF a_eMsgSend[0] = HermesMsgTypeCheckAlive THEN
			fHermesFormCheckAlive(ADR(a_tyXMLTableDataSnd) , p_tyDTStructure , tyCheckAliveSnd);
			fTableConvertToXML(ADR(sSnd) , ADR(udiSndMsgLen) , SIZEOF(sSnd) , ADR(a_tyXMLTableDataSnd) , ADR(a_tyXMLTableDataSnd[0].sTitle) , ADR(a_tyXMLTableDataSnd[0].sValue) , ADR(a_tyXMLTableDataSnd[0].uiSize) , SIZEOF(a_tyXMLTableDataSnd[0]) , 12);

		ELSIF a_eMsgSend[0] = HermesMsgTypeCheckAlivePing THEN
			fHermesFormCheckAlive(ADR(a_tyXMLTableDataSnd) , p_tyDTStructure , tyCheckAlivePingSnd);
			fTableConvertToXML(ADR(sSnd) , ADR(udiSndMsgLen) , SIZEOF(sSnd) , ADR(a_tyXMLTableDataSnd) , ADR(a_tyXMLTableDataSnd[0].sTitle) , ADR(a_tyXMLTableDataSnd[0].sValue) , ADR(a_tyXMLTableDataSnd[0].uiSize) , SIZEOF(a_tyXMLTableDataSnd[0]) , 12);

		ELSIF a_eMsgSend[0] = HermesMsgTypeCheckAlivePong THEN
			fHermesFormCheckAlive(ADR(a_tyXMLTableDataSnd) , p_tyDTStructure , tyCheckAlivePongSnd);
			fTableConvertToXML(ADR(sSnd) , ADR(udiSndMsgLen) , SIZEOF(sSnd) , ADR(a_tyXMLTableDataSnd) , ADR(a_tyXMLTableDataSnd[0].sTitle) , ADR(a_tyXMLTableDataSnd[0].sValue) , ADR(a_tyXMLTableDataSnd[0].uiSize) , SIZEOF(a_tyXMLTableDataSnd[0]) , 12);

		ELSIF a_eMsgSend[0] = HermesMsgTypeServiceDescription THEN
			fHermesFormServiceDescription(ADR(a_tyXMLTableDataSnd) , p_tyDTStructure , tyServiceDescriptionSnd);
			fTableConvertToXML(ADR(sSnd) , ADR(udiSndMsgLen) , SIZEOF(sSnd) , ADR(a_tyXMLTableDataSnd) , ADR(a_tyXMLTableDataSnd[0].sTitle) , ADR(a_tyXMLTableDataSnd[0].sValue) , ADR(a_tyXMLTableDataSnd[0].uiSize) , SIZEOF(a_tyXMLTableDataSnd[0]) , 32); //changed from 30

		ELSIF a_eMsgSend[0] = HermesMsgTypeNotification THEN
			fHermesFormNotification(ADR(a_tyXMLTableDataSnd) , p_tyDTStructure , tyNotificationSnd);
			fTableConvertToXML(ADR(sSnd) , ADR(udiSndMsgLen) , SIZEOF(sSnd) , ADR(a_tyXMLTableDataSnd) , ADR(a_tyXMLTableDataSnd[0].sTitle) , ADR(a_tyXMLTableDataSnd[0].sValue) , ADR(a_tyXMLTableDataSnd[0].uiSize) , SIZEOF(a_tyXMLTableDataSnd[0]) , 14);

		ELSIF a_eMsgSend[0] = HermesMsgTypeBoardAvailable THEN
			eStatus1	:= Error;
			udiStatus1	:= 10135;	//Board Available Request To Send From Upstream Hermes

		ELSIF a_eMsgSend[0] = HermesMsgTypeRevokeBoardAvl THEN
			eStatus1	:= Error;
			udiStatus1	:= 10136;	//Revoke Board Available Request To Send From Upstream Hermes

		ELSIF a_eMsgSend[0] = HermesMsgTypeMachineReady THEN
			fHermesFormMachineReady(ADR(a_tyXMLTableDataSnd) , p_tyDTStructure , tyMachineReady);
			fTableConvertToXML(ADR(sSnd) , ADR(udiSndMsgLen) , SIZEOF(sSnd) , ADR(a_tyXMLTableDataSnd) , ADR(a_tyXMLTableDataSnd[0].sTitle) , ADR(a_tyXMLTableDataSnd[0].sValue) , ADR(a_tyXMLTableDataSnd[0].uiSize) , SIZEOF(a_tyXMLTableDataSnd[0]) , 50);
			bReplyMcRdyId := FALSE;

		ELSIF a_eMsgSend[0] = HermesMsgTypeRevokeMachineReady THEN
			fHermesFormRevokeMachineReady(ADR(a_tyXMLTableDataSnd) , p_tyDTStructure);
			fTableConvertToXML(ADR(sSnd) , ADR(udiSndMsgLen) , SIZEOF(sSnd) , ADR(a_tyXMLTableDataSnd) , ADR(a_tyXMLTableDataSnd[0].sTitle) , ADR(a_tyXMLTableDataSnd[0].sValue) , ADR(a_tyXMLTableDataSnd[0].uiSize) , SIZEOF(a_tyXMLTableDataSnd[0]) , 8);

		ELSIF a_eMsgSend[0] = HermesMsgTypeStartTransport THEN
			fHermesFormStartTransport(ADR(a_tyXMLTableDataSnd) , p_tyDTStructure , tyStartTransport);
			fTableConvertToXML(ADR(sSnd) , ADR(udiSndMsgLen) , SIZEOF(sSnd) , ADR(a_tyXMLTableDataSnd) , ADR(a_tyXMLTableDataSnd[0].sTitle) , ADR(a_tyXMLTableDataSnd[0].sValue) , ADR(a_tyXMLTableDataSnd[0].uiSize) , SIZEOF(a_tyXMLTableDataSnd[0]) , 12);

		ELSIF a_eMsgSend[0] = HermesMsgTypeStopTransport THEN
			fHermesFormStopTransport(ADR(a_tyXMLTableDataSnd) , p_tyDTStructure , tyStopTransport);
			fTableConvertToXML(ADR(sSnd) , ADR(udiSndMsgLen) , SIZEOF(sSnd) , ADR(a_tyXMLTableDataSnd) , ADR(a_tyXMLTableDataSnd[0].sTitle) , ADR(a_tyXMLTableDataSnd[0].sValue) , ADR(a_tyXMLTableDataSnd[0].uiSize) , SIZEOF(a_tyXMLTableDataSnd[0]) , 12);

		ELSIF a_eMsgSend[0] = HermesMsgTypeTransportFinished THEN
			eStatus1	:= Error;
			udiStatus1	:= 10137;	//Transport Finished Request To Send From Upstream Hermes

		ELSIF a_eMsgSend[0] = HermesMsgTypeSetConfiguration THEN
			eStatus1	:= Error;
			udiStatus1	:= 10138;	//Set Configuration Request To Send From Upstream Hermes

		ELSIF a_eMsgSend[0] = HermesMsgTypeGetConfiguration THEN
			eStatus1	:= Error;
			udiStatus1	:= 10139;	//Get Configuration Request To Send From Upstream Hermes

		ELSIF a_eMsgSend[0] = HermesMsgTypeCurrConfiguration THEN
			eStatus1	:= Error;
			udiStatus1	:= 10140;	//Current Configuration Request To Send From Upstream Hermes

		ELSIF a_eMsgSend[0] = HermesMsgTypeBoardForecast THEN
			eStatus1	:= Error;
			udiStatus1	:= 10141;	//Board Forecast Request To Send From Upstream Hermes

		ELSIF a_eMsgSend[0] = HermesMsgTypeQueryBoardInfo THEN
			fHermesFormQueryBoardInfo(ADR(a_tyXMLTableDataSnd) , p_tyDTStructure , tyQueryBoardInfo);
			fTableConvertToXML(ADR(sSnd) , ADR(udiSndMsgLen) , SIZEOF(sSnd) , ADR(a_tyXMLTableDataSnd) , ADR(a_tyXMLTableDataSnd[0].sTitle) , ADR(a_tyXMLTableDataSnd[0].sValue) , ADR(a_tyXMLTableDataSnd[0].uiSize) , SIZEOF(a_tyXMLTableDataSnd[0]) , 12);
			//10142
		ELSIF a_eMsgSend[0] = HermesMsgTypeSendBoardInfo THEN
			eStatus1	:= Error;
			udiStatus1	:= 10159;	//Send Board Info Request To Send From Upstream Hermes

		ELSIF a_eMsgSend[0] = HermesMsgTypeQueryWorkOrderInfo THEN
			eStatus1	:= Error;
			udiStatus1	:= 10160;	//Query Work Order Info Request To Send From Upstream Hermes

		ELSIF a_eMsgSend[0] = HermesMsgTypeSendWorkOrderInfo THEN
			eStatus1	:= Error;
			udiStatus1	:= 10161;	//Send Work Order Info Request To Send From Upstream Hermes

		ELSIF a_eMsgSend[0] = HermesMsgTypeBoardArrived THEN
			eStatus1	:= Error;
			udiStatus1	:= 10162;	//BoardArrived Request To Send From Upstream Hermes

		ELSIF a_eMsgSend[0] = HermesMsgTypeBoardDeparted THEN
			eStatus1	:= Error;
			udiStatus1	:= 10163;	//BoardDeparted Request To Send From Upstream Hermes

		ELSIF a_eMsgSend[0] = HermesMsgTypeCommand THEN
			fHermesFormCommand(ADR(a_tyXMLTableDataSnd) , p_tyDTStructure , tyCommandSnd);
			fTableConvertToXML(ADR(sSnd) , ADR(udiSndMsgLen) , SIZEOF(sSnd) , ADR(a_tyXMLTableDataSnd) , ADR(a_tyXMLTableDataSnd[0].sTitle) , ADR(a_tyXMLTableDataSnd[0].sValue) , ADR(a_tyXMLTableDataSnd[0].uiSize) , SIZEOF(a_tyXMLTableDataSnd[0]) , 10);

		END_IF

		//Message Send
		IF p_bInternalUse = FALSE THEN
			fbSend.udiTCPIdent	:= udiTCPIdent;
			fbSend.udiSndSize	:= udiSndMsgLen;
			fbSend(bEn := TRUE);
		ELSE
			sInternalSnd	:= sSnd;
		END_IF

		IF (fbSend.udiStatus = 0) OR (p_bInternalUse = TRUE) THEN

			fLogDTConvert(ADR(sDT) , p_dtCurrDT);
			memset(ADR(a_sLogList[udiLogCntr]) , 0 , SIZEOF(a_sLogList[udiLogCntr]));
			memcpy(ADR(a_sLogList[udiLogCntr]) + LEN(a_sLogList[udiLogCntr]) , ADR(sDT) , LEN(sDT));
			memcpy(ADR(a_sLogList[udiLogCntr]) + LEN(a_sLogList[udiLogCntr]) , ADR('$r$n') , LEN('$r$n'));
			memcpy(ADR(a_sLogList[udiLogCntr]) + LEN(a_sLogList[udiLogCntr]) , ADR('SND_TO_US$r$n') , LEN('SND_TO_US$r$n'));
			memcpy(ADR(a_sLogList[udiLogCntr]) + LEN(a_sLogList[udiLogCntr]) , ADR(sSnd) , LEN(sSnd));
			memcpy(ADR(a_sLogList[udiLogCntr]) + LEN(a_sLogList[udiLogCntr]) , ADR('$r$n$r$n') , LEN('$r$n$r$n'));

			udiLogCntr	:= udiLogCntr + 1;
			IF udiLogCntr = 11 THEN
				udiLogCntr	:= 1;
			END_IF

			Act_Background_NotificationSnd;
			fHermesRmvOneMsgSend(ADR(a_eMsgSend) , ADR(udiMsgSendBffr));

			fbSend(bEn := FALSE);

		ELSIF (fbSend.udiStatus = 2321) AND (p_bInternalUse = FALSE) THEN
			bRstConnection	:= TRUE;

		ELSIF (fbSend.udiStatus < 65534) AND (p_bInternalUse = FALSE) THEN
			eStatus1	:= Error;

			IF fbSend.udiStatus = 2300 THEN
				udiStatus1	:= 10143;	//Invalid Ident While Sending Data
			ELSIF fbSend.udiStatus = 2320 THEN
				udiStatus1	:= 10144;	//TCP Retry Send Data Error While Sending Data
			ELSIF fbSend.udiStatus = 2322 THEN
				udiStatus1	:= 10145;	//TCP Send Data Error
			ELSE
				udiStatus1	:= fbSend.udiStatus;
			END_IF

		END_IF

	END_IF

END_ACTION
```

#### Act_Background_Err.st - Do Not Change!!!
```iecst
(** 2019-03-15 **)
ACTION Act_Background_Err:

	IF bTransporting = TRUE THEN
		IF bStopTransport AND p_bInterruptSen THEN
			eStatus2	:= Error;
			udiStatus2	:= 10157;	//Board Jam At Sensor After Transfer Interrupted
		END_IF
	END_IF

END_ACTION
```

#### Act_Alarm.st - Do Not Change!!!
```iecst
(** 2021-08-01 **)
ACTION Act_Alarm:

	//Error
	IF EDGEPOS(eStatus = Error) THEN

		tyAlmData.sProgNm		:= p_sProgNm;
		tyAlmData.udiCode		:= udiStatus;
		tyAlmData.eSeverity		:= AlmSeverityError;
		tyAlmData.udiRunTime	:= tyAlmData.udiRunTime + 1;
		tyAlmData.bAlm			:= TRUE;
		tyAlmData.udiModuleNum  := udiModuleNum;
		g_sUSHermesProgNm		:= p_sProgNm;

		//Get Error Message
		IF tyAlmData.udiCode < 10000 OR tyAlmData.udiCode > 10199 THEN
			tyAlmData.sAlmMsg	:= 'Unknown';
			tyAlmData.sRcyMsg	:= 'Unknown';
		ELSE
			tyAlmData.sAlmMsg	:= a_tyAlmText[tyAlmData.udiCode].sAlmText;
			tyAlmData.sRcyMsg	:= a_tyAlmText[tyAlmData.udiCode].sRcyText;
		END_IF

		sStatTxt	:= tyAlmData.sAlmMsg;

	ELSIF bRstErr AND (tyAlmData.udiCode <> 0) THEN

		tyAlmData.udiCode	:= 0;
		tyAlmData.eSeverity	:= AlmSeverityNA;
		tyAlmData.sAlmMsg	:= '';
		tyAlmData.sRcyMsg	:= '';
		tyAlmData.bAlm		:= FALSE;
		sStatTxt	:= a_sStatText[eStat];

	END_IF

END_ACTION
```

#### Act_Alarm2.st - Do Not Change!!!
```iecst
(** 2021-08-01 **)
ACTION Act_Alarm2: //IllegalMsg Check, ChkParamRcv, CmpParamRcv, SequenceTO, B.A Check, B.F Check, bStopTransport

	//Error
	IF EDGEPOS(eStatus2 = Error) THEN

		tyAlmData2.sProgNm		:= p_sProgNm;
		tyAlmData2.udiCode		:= udiStatus2;
		tyAlmData2.eSeverity	:= AlmSeverityError;
		tyAlmData2.udiRunTime	:= tyAlmData2.udiRunTime + 1;
		tyAlmData2.bAlm			:= TRUE;
		tyAlmData2.udiModuleNum := udiModuleNum;
		g_sUSHermesProgNm		:= p_sProgNm;

		//Get Error Message
		IF tyAlmData2.udiCode < 10000 OR tyAlmData2.udiCode > 10199 THEN
			tyAlmData2.sAlmMsg	:= 'Unknown';
			tyAlmData2.sRcyMsg	:= 'Unknown';
		ELSE
			tyAlmData2.sAlmMsg	:= a_tyAlmText[tyAlmData2.udiCode].sAlmText;
			tyAlmData2.sRcyMsg	:= a_tyAlmText[tyAlmData2.udiCode].sRcyText;
		END_IF

		sStatTxt	:= tyAlmData2.sAlmMsg;

	ELSIF bRstErr AND (tyAlmData2.udiCode <> 0) THEN

		tyAlmData2.udiCode		:= 0;
		tyAlmData2.eSeverity	:= AlmSeverityNA;
		tyAlmData2.sAlmMsg		:= '';
		tyAlmData2.sRcyMsg		:= '';
		tyAlmData2.bAlm			:= FALSE;
		sStatTxt	:= a_sStatText[eStat];

	END_IF

END_ACTION
```

#### Act_Alarm3.st - Do Not Change!!!
```iecst
(** 2021-08-01 **)
ACTION Act_Alarm3: //fbFileAppend1 Error

	//Error
	IF EDGEPOS(eStatus3 = Error) THEN

		tyAlmData3.sProgNm		:= p_sProgNm;
		tyAlmData3.udiCode		:= udiStatus3;
		tyAlmData3.eSeverity	:= AlmSeverityError;
		tyAlmData3.udiRunTime	:= tyAlmData3.udiRunTime + 1;
		tyAlmData3.bAlm			:= TRUE;
		tyAlmData3.udiModuleNum := udiModuleNum;
		g_sUSHermesProgNm		:= p_sProgNm;

		//Get Error Message
		IF tyAlmData3.udiCode < 10000 OR tyAlmData3.udiCode > 10199 THEN
			tyAlmData3.sAlmMsg	:= 'Unknown';
			tyAlmData3.sRcyMsg	:= 'Unknown';
		ELSE
			tyAlmData3.sAlmMsg	:= a_tyAlmText[tyAlmData3.udiCode].sAlmText;
			tyAlmData3.sRcyMsg	:= a_tyAlmText[tyAlmData3.udiCode].sRcyText;
		END_IF

		sStatTxt	:= tyAlmData3.sAlmMsg;

	ELSIF bRstErr AND (tyAlmData3.udiCode <> 0) THEN

		tyAlmData3.udiCode		:= 0;
		tyAlmData3.eSeverity	:= AlmSeverityNA;
		tyAlmData3.sAlmMsg		:= '';
		tyAlmData3.sRcyMsg		:= '';
		tyAlmData3.bAlm			:= FALSE;
		sStatTxt	:= a_sStatText[eStat];

	END_IF

END_ACTION
```

#### Act_Alarm4.st - Do Not Change!!!
```iecst
(** 2021-08-01 **)
ACTION Act_Alarm4: //B.A or B.F AccData Error

	//Error
	IF EDGEPOS(eStatus4 = Error) THEN

		tyAlmData4.sProgNm		:= p_sProgNm;
		tyAlmData4.udiCode		:= udiStatus4;
		tyAlmData4.eSeverity	:= AlmSeverityError;
		tyAlmData4.udiRunTime	:= tyAlmData4.udiRunTime + 1;
		tyAlmData4.bAlm			:= TRUE;
		tyAlmData4.udiModuleNum := udiModuleNum;
		g_sUSHermesProgNm		:= p_sProgNm;

		//Get Error Message
		IF tyAlmData4.udiCode < 10000 OR tyAlmData4.udiCode > 10199 THEN
			tyAlmData4.sAlmMsg	:= 'Unknown';
			tyAlmData4.sRcyMsg	:= 'Unknown';
		ELSE
			tyAlmData4.sAlmMsg	:= a_tyAlmText[tyAlmData4.udiCode].sAlmText;
			tyAlmData4.sRcyMsg	:= a_tyAlmText[tyAlmData4.udiCode].sRcyText;
		END_IF

		sStatTxt	:= tyAlmData4.sAlmMsg;

	ELSIF bRstErr AND (tyAlmData4.udiCode <> 0) THEN

		tyAlmData4.udiCode		:= 0;
		tyAlmData4.eSeverity	:= AlmSeverityNA;
		tyAlmData4.sAlmMsg		:= '';
		tyAlmData4.sRcyMsg		:= '';
		tyAlmData4.bAlm			:= FALSE;
		sStatTxt	:= a_sStatText[eStat];

	END_IF

END_ACTION
```
